KUKA KRL program: f1_Kuka_APT212T03S12.SRC

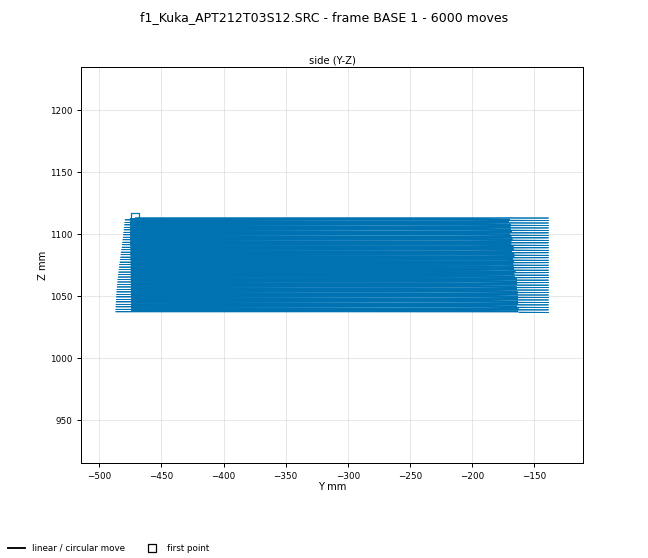
[picture p0: tool path of f1_Kuka_APT212T03S12.SRC in frame BASE 1, 6000 of 6001 moves have a stored position in this frame; points joined in program order, loops and branches not executed]
&ACCESS RVP
&REL 2
&PARAM TEMPLATE = C:\KRC\Roboter\Template\vorgabe
&PARAM EDITMASK = *
DEF f1_Kuka_APT212T03S12()


;FOLD INI;%{PE}%V3.2.0,%MKUKATPBASIS,%CINIT,%VCOMMON,%P
  ;FOLD BAS INI;%{E}%V3.2.0,%MKUKATPBASIS,%CINIT,%VINIT,%P
    GLOBAL INTERRUPT DECL 3 WHEN $STOPMESS==TRUE DO IR_STOPM ( )
    INTERRUPT ON 3
    BAS (#INITMOV,0 )
  ;ENDFOLD (BAS INI)
  ;FOLD USER INI;%{E}%V3.2.0,%MKUKATPUSER,%CINIT,%VINIT,%P
    ;Make your modifications here
  ;ENDFOLD (USER INI)
;ENDFOLD (INI)


;*** Make Null PTP Move
  PTP $pos_act

;*** Auto Load The Correct TOOL Data
  $tool=tool_data[3]

;*** Auto Load The Correct BASE Data
  $base=base_data[1]

  $ADVANCE = 5

;*** Restate Last Velocity
MMPM(30000.0)
SetRPM(6000)
LIN {X -0.139,Y -471.059,Z 1113.517,A 0.000,B 0.000,C 90.000,E1 273.151} C_DIS
LIN {X -0.055,Y -467.604,Z 1113.515,A 0.000,B 0.000,C 90.000,E1 272.636} C_DIS
LIN {X 0.015,Y -463.098,Z 1113.512,A 0.000,B 0.000,C 90.000,E1 272.121} C_DIS
LIN {X 0.076,Y -457.357,Z 1113.509,A 0.000,B 0.000,C 90.000,E1 271.604} C_DIS
LIN {X 0.094,Y -450.718,Z 1113.506,A 0.000,B 0.000,C 90.000,E1 271.146} C_DIS
LIN {X -0.014,Y -447.591,Z 1113.505,A 0.000,B 0.000,C 90.000,E1 270.974} C_DIS
LIN {X 0.034,Y -440.708,Z 1113.504,A 0.000,B 0.000,C 90.000,E1 270.630} C_DIS
LIN {X 0.083,Y -433.709,Z 1113.502,A 0.000,B 0.000,C 90.000,E1 270.344} C_DIS
LIN {X 0.062,Y -426.679,Z 1113.501,A 0.000,B 0.000,C 90.000,E1 270.115} C_DIS
LIN {X -0.084,Y -419.545,Z 1113.500,A 0.000,B 0.000,C 90.000,E1 269.943} C_DIS
LIN {X 0.009,Y -412.022,Z 1113.499,A 0.000,B 0.000,C 90.000,E1 269.771} C_DIS
LIN {X -0.097,Y -403.841,Z 1113.498,A 0.000,B 0.000,C 90.000,E1 269.656} C_DIS
LIN {X 0.016,Y -391.803,Z 1113.497,A 0.000,B 0.000,C 90.000,E1 269.542} C_DIS
LIN {X -0.051,Y -388.701,Z 1113.497,A 0.000,B 0.000,C 90.000,E1 269.542} C_DIS
LIN {X -0.056,Y -181.444,Z 1113.497,A 0.000,B 0.000,C 90.000,E1 269.542} C_DIS
LIN {X -0.018,Y -180.903,Z 1113.474,A 0.000,B 0.000,C 90.000,E1 265.298} C_DIS
LIN {X -0.068,Y -180.241,Z 1113.464,A 0.000,B 0.000,C 90.000,E1 263.628} C_DIS
LIN {X -0.049,Y -178.727,Z 1113.441,A 0.000,B 0.000,C 90.000,E1 259.398} C_DIS
LIN {X 0.018,Y -175.775,Z 1113.413,A 0.000,B 0.000,C 90.000,E1 254.283} C_DIS
LIN {X 0.006,Y -171.960,Z 1113.384,A 0.000,B 0.000,C 90.000,E1 249.156} C_DIS
LIN {X 0.044,Y -171.353,Z 1113.379,A 0.000,B 0.000,C 90.000,E1 248.284} C_DIS
LIN {X 0.021,Y -167.603,Z 1113.355,A 0.000,B 0.000,C 90.000,E1 243.973} C_DIS
LIN {X 0.034,Y -166.248,Z 1113.346,A 0.000,B 0.000,C 90.000,E1 242.231} C_DIS
LIN {X 0.021,Y -163.004,Z 1113.326,A 0.000,B 0.000,C 90.000,E1 238.742} C_DIS
LIN {X 0.068,Y -160.925,Z 1113.312,A 0.000,B 0.000,C 90.000,E1 236.087} C_DIS
LIN {X 0.045,Y -157.686,Z 1113.292,A 0.000,B 0.000,C 90.000,E1 232.557} C_DIS
LIN {X -0.016,Y -155.726,Z 1113.277,A 0.000,B 0.000,C 90.000,E1 229.908} C_DIS
LIN {X 0.037,Y -151.985,Z 1113.252,A 0.000,B 0.000,C 90.000,E1 225.405} C_DIS
LIN {X 0.053,Y -150.230,Z 1113.237,A 0.000,B 0.000,C 90.000,E1 222.690} C_DIS
LIN {X -0.024,Y -146.991,Z 1113.212,A 0.000,B 0.000,C 90.000,E1 218.177} C_DIS
LIN {X -0.033,Y -145.576,Z 1113.197,A 0.000,B 0.000,C 90.000,E1 215.438} C_DIS
LIN {X 0.083,Y -142.965,Z 1113.171,A 0.000,B 0.000,C 90.000,E1 210.797} C_DIS
LIN {X 0.013,Y -141.593,Z 1113.151,A 0.000,B 0.000,C 90.000,E1 207.129} C_DIS
LIN {X 0.061,Y -139.420,Z 1113.115,A 0.000,B 0.000,C 90.000,E1 200.610} C_DIS
LIN {X -0.019,Y -139.147,Z 1113.104,A 0.000,B 0.000,C 90.000,E1 198.779} C_DIS
LIN {X 0.003,Y -138.346,Z 1113.058,A 0.000,B 0.000,C 90.000,E1 190.366} C_DIS
LIN {X -0.011,Y -139.488,Z 1113.006,A 0.000,B 0.000,C 90.000,E1 181.031} C_DIS
LIN {X -0.071,Y -141.091,Z 1112.975,A 0.000,B 0.000,C 90.000,E1 175.469} C_DIS
LIN {X 0.023,Y -142.469,Z 1112.959,A 0.000,B 0.000,C 90.000,E1 172.648} C_DIS
LIN {X -0.029,Y -144.715,Z 1112.934,A 0.000,B 0.000,C 90.000,E1 168.049} C_DIS
LIN {X 0.064,Y -147.315,Z 1112.913,A 0.000,B 0.000,C 90.000,E1 164.338} C_DIS
LIN {X -0.063,Y -150.636,Z 1112.888,A 0.000,B 0.000,C 90.000,E1 159.826} C_DIS
LIN {X 0.012,Y -154.113,Z 1112.868,A 0.000,B 0.000,C 90.000,E1 156.177} C_DIS
LIN {X -0.064,Y -157.538,Z 1112.848,A 0.000,B 0.000,C 90.000,E1 152.615} C_DIS
LIN {X 0.101,Y -161.775,Z 1112.828,A 0.000,B 0.000,C 90.000,E1 148.997} C_DIS
LIN {X -0.014,Y -165.968,Z 1112.808,A 0.000,B 0.000,C 90.000,E1 145.515} C_DIS
LIN {X -0.019,Y -170.962,Z 1112.789,A 0.000,B 0.000,C 90.000,E1 142.029} C_DIS
LIN {X 0.033,Y -175.831,Z 1112.770,A 0.000,B 0.000,C 90.000,E1 138.566} C_DIS
LIN {X 0.028,Y -181.437,Z 1112.751,A 0.000,B 0.000,C 90.000,E1 135.162} C_DIS
LIN {X -0.098,Y -186.943,Z 1112.732,A 0.000,B 0.000,C 90.000,E1 131.838} C_DIS
LIN {X -0.100,Y -190.056,Z 1112.723,A 0.000,B 0.000,C 90.000,E1 130.172} C_DIS
LIN {X -0.085,Y -195.830,Z 1112.705,A 0.000,B 0.000,C 90.000,E1 126.870} C_DIS
LIN {X 0.022,Y -200.393,Z 1112.692,A 0.000,B 0.000,C 90.000,E1 124.532} C_DIS
LIN {X -0.001,Y -308.324,Z 1112.692,A 0.000,B 0.000,C 90.000,E1 124.532} C_DIS
LIN {X -0.072,Y -309.497,Z 1112.692,A 0.000,B 0.000,C 90.000,E1 124.532} C_DIS
LIN {X -0.028,Y -313.075,Z 1112.691,A 0.000,B 0.000,C 90.000,E1 124.405} C_DIS
LIN {X -0.040,Y -316.216,Z 1112.690,A 0.000,B 0.000,C 90.000,E1 124.199} C_DIS
LIN {X 0.038,Y -319.912,Z 1112.688,A 0.000,B 0.000,C 90.000,E1 123.785} C_DIS
LIN {X -0.021,Y -321.827,Z 1112.686,A 0.000,B 0.000,C 90.000,E1 123.499} C_DIS
LIN {X -0.081,Y -323.333,Z 1112.684,A 0.000,B 0.000,C 90.000,E1 123.214} C_DIS
LIN {X -0.084,Y -326.852,Z 1112.679,A 0.000,B 0.000,C 90.000,E1 122.260} C_DIS
LIN {X 0.052,Y -337.735,Z 1112.663,A 0.000,B 0.000,C 90.000,E1 119.411} C_DIS
LIN {X -0.122,Y -349.996,Z 1112.648,A 0.000,B 0.000,C 90.000,E1 116.668} C_DIS
LIN {X -0.116,Y -363.748,Z 1112.633,A 0.000,B 0.000,C 90.000,E1 113.951} C_DIS
LIN {X -0.114,Y -377.318,Z 1112.620,A 0.000,B 0.000,C 90.000,E1 111.589} C_DIS
LIN {X -0.044,Y -392.255,Z 1112.607,A 0.000,B 0.000,C 90.000,E1 109.268} C_DIS
LIN {X 0.158,Y -408.666,Z 1112.594,A 0.000,B 0.000,C 90.000,E1 106.985} C_DIS
LIN {X -0.146,Y -426.666,Z 1112.582,A 0.000,B 0.000,C 90.000,E1 104.828} C_DIS
LIN {X -0.136,Y -446.228,Z 1112.570,A 0.000,B 0.000,C 90.000,E1 102.703} C_DIS
LIN {X 0.014,Y -468.953,Z 1112.558,A 0.000,B 0.000,C 90.000,E1 100.489} C_DIS
LIN {X 0.041,Y -470.834,Z 1112.557,A 0.000,B 0.000,C 90.000,E1 100.254} C_DIS
LIN {X -0.107,Y -472.388,Z 1112.556,A 0.000,B 0.000,C 90.000,E1 100.018} C_DIS
LIN {X 0.211,Y -473.550,Z 1112.554,A 0.000,B 0.000,C 90.000,E1 99.726} C_DIS
LIN {X -0.147,Y -474.953,Z 1112.551,A 0.000,B 0.000,C 90.000,E1 99.265} C_DIS
LIN {X -0.026,Y -475.327,Z 1112.549,A 0.000,B 0.000,C 90.000,E1 98.746} C_DIS
LIN {X 0.173,Y -474.738,Z 1112.546,A 0.000,B 0.000,C 90.000,E1 98.219} C_DIS
LIN {X -0.166,Y -473.095,Z 1112.543,A 0.000,B 0.000,C 90.000,E1 97.757} C_DIS
LIN {X 0.102,Y -471.788,Z 1112.542,A 0.000,B 0.000,C 90.000,E1 97.473} C_DIS
LIN {X 0.009,Y -457.406,Z 1112.530,A 0.000,B 0.000,C 90.000,E1 95.454} C_DIS
LIN {X -0.050,Y -439.778,Z 1112.516,A 0.000,B 0.000,C 90.000,E1 92.865} C_DIS
LIN {X -0.072,Y -426.758,Z 1112.504,A 0.000,B 0.000,C 90.000,E1 90.745} C_DIS
LIN {X -0.028,Y -408.534,Z 1112.486,A 0.000,B 0.000,C 90.000,E1 87.478} C_DIS
LIN {X -0.013,Y -399.508,Z 1112.477,A 0.000,B 0.000,C 90.000,E1 85.812} C_DIS
LIN {X -0.106,Y -388.900,Z 1112.466,A 0.000,B 0.000,C 90.000,E1 83.856} C_DIS
LIN {X -0.001,Y -378.381,Z 1112.455,A 0.000,B 0.000,C 90.000,E1 81.837} C_DIS
LIN {X -0.006,Y -369.144,Z 1112.445,A 0.000,B 0.000,C 90.000,E1 80.095} C_DIS
LIN {X -0.108,Y -359.479,Z 1112.435,A 0.000,B 0.000,C 90.000,E1 78.342} C_DIS
LIN {X 0.042,Y -349.580,Z 1112.425,A 0.000,B 0.000,C 90.000,E1 76.520} C_DIS
LIN {X -0.003,Y -338.018,Z 1112.413,A 0.000,B 0.000,C 90.000,E1 74.393} C_DIS
LIN {X 0.018,Y -323.542,Z 1112.398,A 0.000,B 0.000,C 90.000,E1 71.583} C_DIS
LIN {X -0.047,Y -309.901,Z 1112.382,A 0.000,B 0.000,C 90.000,E1 68.720} C_DIS
LIN {X -0.139,Y -297.027,Z 1112.365,A 0.000,B 0.000,C 90.000,E1 65.793} C_DIS
LIN {X 0.053,Y -284.665,Z 1112.349,A 0.000,B 0.000,C 90.000,E1 62.743} C_DIS
LIN {X 0.089,Y -274.024,Z 1112.333,A 0.000,B 0.000,C 90.000,E1 59.999} C_DIS
LIN {X -0.096,Y -263.649,Z 1112.318,A 0.000,B 0.000,C 90.000,E1 57.248} C_DIS
LIN {X 0.013,Y -251.356,Z 1112.298,A 0.000,B 0.000,C 90.000,E1 53.657} C_DIS
LIN {X 0.084,Y -240.974,Z 1112.280,A 0.000,B 0.000,C 90.000,E1 50.356} C_DIS
LIN {X 0.013,Y -231.416,Z 1112.261,A 0.000,B 0.000,C 90.000,E1 47.025} C_DIS
LIN {X 0.072,Y -221.510,Z 1112.240,A 0.000,B 0.000,C 90.000,E1 43.218} C_DIS
LIN {X 0.029,Y -212.142,Z 1112.219,A 0.000,B 0.000,C 90.000,E1 39.358} C_DIS
LIN {X -0.011,Y -205.168,Z 1112.201,A 0.000,B 0.000,C 90.000,E1 36.217} C_DIS
LIN {X 0.026,Y -198.680,Z 1112.183,A 0.000,B 0.000,C 90.000,E1 33.007} C_DIS
LIN {X -0.084,Y -192.840,Z 1112.165,A 0.000,B 0.000,C 90.000,E1 29.795} C_DIS
LIN {X -0.018,Y -187.519,Z 1112.147,A 0.000,B 0.000,C 90.000,E1 26.488} C_DIS
LIN {X 0.012,Y -182.914,Z 1112.129,A 0.000,B 0.000,C 90.000,E1 23.153} C_DIS
LIN {X -0.046,Y -179.023,Z 1112.110,A 0.000,B 0.000,C 90.000,E1 19.812} C_DIS
LIN {X 0.012,Y -175.068,Z 1112.086,A 0.000,B 0.000,C 90.000,E1 15.552} C_DIS
LIN {X -0.065,Y -172.119,Z 1112.063,A 0.000,B 0.000,C 90.000,E1 11.299} C_DIS
LIN {X 0.069,Y -169.810,Z 1112.029,A 0.000,B 0.000,C 90.000,E1 5.220} C_DIS
LIN {X 0.050,Y -170.803,Z 1111.964,A 0.000,B 0.000,C 90.000,E1 353.457} C_DIS
LIN {X 0.054,Y -173.493,Z 1111.935,A 0.000,B 0.000,C 90.000,E1 348.285} C_DIS
LIN {X -0.029,Y -176.809,Z 1111.911,A 0.000,B 0.000,C 90.000,E1 344.031} C_DIS
LIN {X 0.071,Y -181.080,Z 1111.888,A 0.000,B 0.000,C 90.000,E1 339.752} C_DIS
LIN {X -0.005,Y -185.214,Z 1111.869,A 0.000,B 0.000,C 90.000,E1 336.410} C_DIS
LIN {X -0.007,Y -190.069,Z 1111.850,A 0.000,B 0.000,C 90.000,E1 333.076} C_DIS
LIN {X -0.055,Y -195.639,Z 1111.832,A 0.000,B 0.000,C 90.000,E1 329.793} C_DIS
LIN {X 0.072,Y -201.884,Z 1111.814,A 0.000,B 0.000,C 90.000,E1 326.501} C_DIS
LIN {X -0.094,Y -208.900,Z 1111.796,A 0.000,B 0.000,C 90.000,E1 323.336} C_DIS
LIN {X -0.005,Y -216.661,Z 1111.779,A 0.000,B 0.000,C 90.000,E1 320.150} C_DIS
LIN {X -0.078,Y -225.301,Z 1111.761,A 0.000,B 0.000,C 90.000,E1 317.067} C_DIS
LIN {X -0.102,Y -235.017,Z 1111.745,A 0.000,B 0.000,C 90.000,E1 314.028} C_DIS
LIN {X -0.003,Y -244.461,Z 1111.730,A 0.000,B 0.000,C 90.000,E1 311.391} C_DIS
LIN {X -0.029,Y -253.486,Z 1111.718,A 0.000,B 0.000,C 90.000,E1 309.197} C_DIS
LIN {X 0.046,Y -265.217,Z 1111.704,A 0.000,B 0.000,C 90.000,E1 306.664} C_DIS
LIN {X 0.120,Y -281.653,Z 1111.686,A 0.000,B 0.000,C 90.000,E1 303.499} C_DIS
LIN {X 0.046,Y -297.378,Z 1111.671,A 0.000,B 0.000,C 90.000,E1 300.797} C_DIS
LIN {X -0.029,Y -316.878,Z 1111.655,A 0.000,B 0.000,C 90.000,E1 297.847} C_DIS
LIN {X 0.057,Y -335.880,Z 1111.641,A 0.000,B 0.000,C 90.000,E1 295.283} C_DIS
LIN {X 0.015,Y -351.312,Z 1111.630,A 0.000,B 0.000,C 90.000,E1 293.462} C_DIS
LIN {X 0.107,Y -367.275,Z 1111.621,A 0.000,B 0.000,C 90.000,E1 291.770} C_DIS
LIN {X 0.039,Y -392.129,Z 1111.608,A 0.000,B 0.000,C 90.000,E1 289.504} C_DIS
LIN {X 0.001,Y -405.648,Z 1111.602,A 0.000,B 0.000,C 90.000,E1 288.308} C_DIS
LIN {X 0.092,Y -416.173,Z 1111.596,A 0.000,B 0.000,C 90.000,E1 287.330} C_DIS
LIN {X -0.150,Y -423.969,Z 1111.592,A 0.000,B 0.000,C 90.000,E1 286.622} C_DIS
LIN {X -0.028,Y -431.548,Z 1111.588,A 0.000,B 0.000,C 90.000,E1 285.843} C_DIS
LIN {X -0.081,Y -438.876,Z 1111.584,A 0.000,B 0.000,C 90.000,E1 285.064} C_DIS
LIN {X 0.109,Y -445.762,Z 1111.579,A 0.000,B 0.000,C 90.000,E1 284.245} C_DIS
LIN {X -0.063,Y -452.032,Z 1111.575,A 0.000,B 0.000,C 90.000,E1 283.480} C_DIS
LIN {X -0.088,Y -457.614,Z 1111.571,A 0.000,B 0.000,C 90.000,E1 282.703} C_DIS
LIN {X -0.261,Y -462.481,Z 1111.566,A 0.000,B 0.000,C 90.000,E1 281.951} C_DIS
LIN {X 0.159,Y -466.725,Z 1111.562,A 0.000,B 0.000,C 90.000,E1 281.130} C_DIS
LIN {X 0.163,Y -470.343,Z 1111.558,A 0.000,B 0.000,C 90.000,E1 280.366} C_DIS
LIN {X 0.109,Y -473.331,Z 1111.553,A 0.000,B 0.000,C 90.000,E1 279.613} C_DIS
LIN {X -0.253,Y -475.008,Z 1111.551,A 0.000,B 0.000,C 90.000,E1 279.151} C_DIS
LIN {X -0.062,Y -476.427,Z 1111.548,A 0.000,B 0.000,C 90.000,E1 278.624} C_DIS
LIN {X 0.068,Y -477.604,Z 1111.545,A 0.000,B 0.000,C 90.000,E1 278.106} C_DIS
LIN {X 0.208,Y -478.452,Z 1111.542,A 0.000,B 0.000,C 90.000,E1 277.587} C_DIS
LIN {X -0.118,Y -479.069,Z 1111.540,A 0.000,B 0.000,C 90.000,E1 277.125} C_DIS
LIN {X 0.037,Y -479.395,Z 1111.537,A 0.000,B 0.000,C 90.000,E1 276.606} C_DIS
LIN {X 0.195,Y -479.403,Z 1111.534,A 0.000,B 0.000,C 90.000,E1 276.087} C_DIS
LIN {X -0.122,Y -479.104,Z 1111.531,A 0.000,B 0.000,C 90.000,E1 275.625} C_DIS
LIN {X 0.037,Y -478.438,Z 1111.528,A 0.000,B 0.000,C 90.000,E1 275.106} C_DIS
LIN {X 0.191,Y -477.392,Z 1111.526,A 0.000,B 0.000,C 90.000,E1 274.588} C_DIS
LIN {X -0.170,Y -475.931,Z 1111.523,A 0.000,B 0.000,C 90.000,E1 274.131} C_DIS
LIN {X -0.027,Y -473.925,Z 1111.520,A 0.000,B 0.000,C 90.000,E1 273.612} C_DIS
LIN {X 0.103,Y -471.258,Z 1111.517,A 0.000,B 0.000,C 90.000,E1 273.094} C_DIS
LIN {X 0.187,Y -467.779,Z 1111.514,A 0.000,B 0.000,C 90.000,E1 272.579} C_DIS
LIN {X -0.011,Y -465.688,Z 1111.513,A 0.000,B 0.000,C 90.000,E1 272.350} C_DIS
LIN {X -0.207,Y -463.300,Z 1111.512,A 0.000,B 0.000,C 90.000,E1 272.121} C_DIS
LIN {X -0.142,Y -457.521,Z 1111.509,A 0.000,B 0.000,C 90.000,E1 271.604} C_DIS
LIN {X -0.080,Y -450.984,Z 1111.506,A 0.000,B 0.000,C 90.000,E1 271.146} C_DIS
LIN {X -0.200,Y -447.827,Z 1111.505,A 0.000,B 0.000,C 90.000,E1 270.974} C_DIS
LIN {X -0.172,Y -440.828,Z 1111.503,A 0.000,B 0.000,C 90.000,E1 270.630} C_DIS
LIN {X -0.140,Y -433.831,Z 1111.502,A 0.000,B 0.000,C 90.000,E1 270.344} C_DIS
LIN {X -0.148,Y -426.727,Z 1111.500,A 0.000,B 0.000,C 90.000,E1 270.115} C_DIS
LIN {X 0.155,Y -419.712,Z 1111.500,A 0.000,B 0.000,C 90.000,E1 269.885} C_DIS
LIN {X 0.185,Y -408.271,Z 1111.498,A 0.000,B 0.000,C 90.000,E1 269.656} C_DIS
LIN {X 0.035,Y -395.985,Z 1111.497,A 0.000,B 0.000,C 90.000,E1 269.542} C_DIS
LIN {X -0.169,Y -387.727,Z 1111.497,A 0.000,B 0.000,C 90.000,E1 269.542} C_DIS
LIN {X 0.071,Y -181.441,Z 1111.497,A 0.000,B 0.000,C 90.000,E1 269.484} C_DIS
LIN {X -0.073,Y -180.903,Z 1111.474,A 0.000,B 0.000,C 90.000,E1 265.298} C_DIS
LIN {X 0.057,Y -180.233,Z 1111.464,A 0.000,B 0.000,C 90.000,E1 263.571} C_DIS
LIN {X 0.072,Y -178.717,Z 1111.441,A 0.000,B 0.000,C 90.000,E1 259.342} C_DIS
LIN {X -0.035,Y -175.765,Z 1111.413,A 0.000,B 0.000,C 90.000,E1 254.283} C_DIS
LIN {X 0.014,Y -171.949,Z 1111.384,A 0.000,B 0.000,C 90.000,E1 249.135} C_DIS
LIN {X -0.009,Y -171.337,Z 1111.379,A 0.000,B 0.000,C 90.000,E1 248.284} C_DIS
LIN {X -0.031,Y -167.591,Z 1111.355,A 0.000,B 0.000,C 90.000,E1 243.973} C_DIS
LIN {X -0.018,Y -166.229,Z 1111.346,A 0.000,B 0.000,C 90.000,E1 242.231} C_DIS
LIN {X -0.030,Y -162.989,Z 1111.326,A 0.000,B 0.000,C 90.000,E1 238.742} C_DIS
LIN {X 0.017,Y -160.907,Z 1111.312,A 0.000,B 0.000,C 90.000,E1 236.087} C_DIS
LIN {X -0.005,Y -157.672,Z 1111.292,A 0.000,B 0.000,C 90.000,E1 232.557} C_DIS
LIN {X -0.067,Y -155.711,Z 1111.277,A 0.000,B 0.000,C 90.000,E1 229.908} C_DIS
LIN {X -0.013,Y -151.972,Z 1111.252,A 0.000,B 0.000,C 90.000,E1 225.405} C_DIS
LIN {X 0.005,Y -150.215,Z 1111.237,A 0.000,B 0.000,C 90.000,E1 222.690} C_DIS
LIN {X -0.072,Y -146.980,Z 1111.212,A 0.000,B 0.000,C 90.000,E1 218.177} C_DIS
LIN {X 0.037,Y -145.567,Z 1111.197,A 0.000,B 0.000,C 90.000,E1 215.391} C_DIS
LIN {X 0.037,Y -142.957,Z 1111.171,A 0.000,B 0.000,C 90.000,E1 210.797} C_DIS
LIN {X -0.033,Y -141.584,Z 1111.151,A 0.000,B 0.000,C 90.000,E1 207.129} C_DIS
LIN {X 0.014,Y -139.417,Z 1111.115,A 0.000,B 0.000,C 90.000,E1 200.610} C_DIS
LIN {X 0.067,Y -139.142,Z 1111.104,A 0.000,B 0.000,C 90.000,E1 198.725} C_DIS
LIN {X -0.043,Y -138.347,Z 1111.057,A 0.000,B 0.000,C 90.000,E1 190.366} C_DIS
LIN {X -0.058,Y -139.491,Z 1111.006,A 0.000,B 0.000,C 90.000,E1 181.031} C_DIS
LIN {X 0.023,Y -141.099,Z 1110.975,A 0.000,B 0.000,C 90.000,E1 175.412} C_DIS
LIN {X -0.024,Y -142.479,Z 1110.959,A 0.000,B 0.000,C 90.000,E1 172.648} C_DIS
LIN {X 0.065,Y -144.727,Z 1110.933,A 0.000,B 0.000,C 90.000,E1 167.993} C_DIS
LIN {X 0.016,Y -147.330,Z 1110.913,A 0.000,B 0.000,C 90.000,E1 164.338} C_DIS
LIN {X 0.081,Y -150.652,Z 1110.888,A 0.000,B 0.000,C 90.000,E1 159.752} C_DIS
LIN {X -0.037,Y -154.130,Z 1110.868,A 0.000,B 0.000,C 90.000,E1 156.177} C_DIS
LIN {X 0.025,Y -157.557,Z 1110.848,A 0.000,B 0.000,C 90.000,E1 152.564} C_DIS
LIN {X 0.050,Y -161.799,Z 1110.828,A 0.000,B 0.000,C 90.000,E1 148.997} C_DIS
LIN {X 0.070,Y -165.990,Z 1110.808,A 0.000,B 0.000,C 90.000,E1 145.468} C_DIS
LIN {X 0.063,Y -170.989,Z 1110.789,A 0.000,B 0.000,C 90.000,E1 141.984} C_DIS
LIN {X -0.021,Y -175.857,Z 1110.770,A 0.000,B 0.000,C 90.000,E1 138.566} C_DIS
LIN {X -0.027,Y -181.463,Z 1110.751,A 0.000,B 0.000,C 90.000,E1 135.162} C_DIS
LIN {X 0.110,Y -186.974,Z 1110.732,A 0.000,B 0.000,C 90.000,E1 131.757} C_DIS
LIN {X 0.112,Y -190.088,Z 1110.723,A 0.000,B 0.000,C 90.000,E1 130.092} C_DIS
LIN {X 0.015,Y -195.861,Z 1110.705,A 0.000,B 0.000,C 90.000,E1 126.824} C_DIS
LIN {X 0.017,Y -200.329,Z 1110.692,A 0.000,B 0.000,C 90.000,E1 124.565} C_DIS
LIN {X 0.166,Y -307.637,Z 1110.692,A 0.000,B 0.000,C 90.000,E1 124.532} C_DIS
LIN {X 0.131,Y -308.781,Z 1110.692,A 0.000,B 0.000,C 90.000,E1 124.532} C_DIS
LIN {X -0.118,Y -313.804,Z 1110.691,A 0.000,B 0.000,C 90.000,E1 124.405} C_DIS
LIN {X -0.174,Y -316.709,Z 1110.690,A 0.000,B 0.000,C 90.000,E1 124.199} C_DIS
LIN {X 0.113,Y -320.458,Z 1110.687,A 0.000,B 0.000,C 90.000,E1 123.706} C_DIS
LIN {X -0.049,Y -322.322,Z 1110.686,A 0.000,B 0.000,C 90.000,E1 123.420} C_DIS
LIN {X 0.056,Y -323.778,Z 1110.684,A 0.000,B 0.000,C 90.000,E1 123.086} C_DIS
LIN {X 0.082,Y -336.846,Z 1110.665,A 0.000,B 0.000,C 90.000,E1 119.617} C_DIS
LIN {X -0.115,Y -349.001,Z 1110.649,A 0.000,B 0.000,C 90.000,E1 116.873} C_DIS
LIN {X 0.024,Y -362.634,Z 1110.634,A 0.000,B 0.000,C 90.000,E1 114.131} C_DIS
LIN {X 0.000,Y -376.093,Z 1110.621,A 0.000,B 0.000,C 90.000,E1 111.770} C_DIS
LIN {X 0.040,Y -390.910,Z 1110.608,A 0.000,B 0.000,C 90.000,E1 109.450} C_DIS
LIN {X -0.178,Y -407.190,Z 1110.596,A 0.000,B 0.000,C 90.000,E1 107.221} C_DIS
LIN {X -0.123,Y -425.050,Z 1110.583,A 0.000,B 0.000,C 90.000,E1 105.009} C_DIS
LIN {X -0.179,Y -444.502,Z 1110.571,A 0.000,B 0.000,C 90.000,E1 102.883} C_DIS
LIN {X -0.085,Y -464.739,Z 1110.560,A 0.000,B 0.000,C 90.000,E1 100.894} C_DIS
LIN {X -0.060,Y -469.593,Z 1110.558,A 0.000,B 0.000,C 90.000,E1 100.423} C_DIS
LIN {X -0.111,Y -471.308,Z 1110.557,A 0.000,B 0.000,C 90.000,E1 100.197} C_DIS
LIN {X 0.209,Y -472.734,Z 1110.555,A 0.000,B 0.000,C 90.000,E1 99.905} C_DIS
LIN {X 0.063,Y -473.796,Z 1110.554,A 0.000,B 0.000,C 90.000,E1 99.670} C_DIS
LIN {X 0.176,Y -475.035,Z 1110.551,A 0.000,B 0.000,C 90.000,E1 99.151} C_DIS
LIN {X -0.098,Y -475.268,Z 1110.548,A 0.000,B 0.000,C 90.000,E1 98.681} C_DIS
LIN {X 0.029,Y -474.534,Z 1110.545,A 0.000,B 0.000,C 90.000,E1 98.163} C_DIS
LIN {X 0.161,Y -472.714,Z 1110.543,A 0.000,B 0.000,C 90.000,E1 97.644} C_DIS
LIN {X 0.022,Y -471.293,Z 1110.541,A 0.000,B 0.000,C 90.000,E1 97.409} C_DIS
LIN {X -0.094,Y -456.843,Z 1110.530,A 0.000,B 0.000,C 90.000,E1 95.391} C_DIS
LIN {X 0.057,Y -440.932,Z 1110.517,A 0.000,B 0.000,C 90.000,E1 93.037} C_DIS
LIN {X 0.056,Y -427.874,Z 1110.505,A 0.000,B 0.000,C 90.000,E1 90.917} C_DIS
LIN {X -0.147,Y -413.962,Z 1110.492,A 0.000,B 0.000,C 90.000,E1 88.511} C_DIS
LIN {X -0.039,Y -405.097,Z 1110.482,A 0.000,B 0.000,C 90.000,E1 86.846} C_DIS
LIN {X -0.047,Y -394.489,Z 1110.472,A 0.000,B 0.000,C 90.000,E1 84.894} C_DIS
LIN {X 0.162,Y -382.415,Z 1110.459,A 0.000,B 0.000,C 90.000,E1 82.591} C_DIS
LIN {X -0.146,Y -373.276,Z 1110.449,A 0.000,B 0.000,C 90.000,E1 80.905} C_DIS
LIN {X 0.138,Y -365.409,Z 1110.441,A 0.000,B 0.000,C 90.000,E1 79.398} C_DIS
LIN {X 0.007,Y -357.267,Z 1110.433,A 0.000,B 0.000,C 90.000,E1 77.937} C_DIS
LIN {X 0.032,Y -345.686,Z 1110.421,A 0.000,B 0.000,C 90.000,E1 75.825} C_DIS
LIN {X -0.016,Y -334.165,Z 1110.409,A 0.000,B 0.000,C 90.000,E1 73.685} C_DIS
LIN {X -0.059,Y -318.384,Z 1110.392,A 0.000,B 0.000,C 90.000,E1 70.550} C_DIS
LIN {X 0.050,Y -302.190,Z 1110.372,A 0.000,B 0.000,C 90.000,E1 66.975} C_DIS
LIN {X -0.127,Y -289.617,Z 1110.356,A 0.000,B 0.000,C 90.000,E1 64.024} C_DIS
LIN {X 0.106,Y -277.484,Z 1110.339,A 0.000,B 0.000,C 90.000,E1 60.923} C_DIS
LIN {X -0.135,Y -266.989,Z 1110.323,A 0.000,B 0.000,C 90.000,E1 58.201} C_DIS
LIN {X 0.084,Y -254.446,Z 1110.303,A 0.000,B 0.000,C 90.000,E1 54.609} C_DIS
LIN {X -0.049,Y -243.833,Z 1110.285,A 0.000,B 0.000,C 90.000,E1 51.376} C_DIS
LIN {X 0.011,Y -235.060,Z 1110.269,A 0.000,B 0.000,C 90.000,E1 48.405} C_DIS
LIN {X -0.128,Y -224.893,Z 1110.248,A 0.000,B 0.000,C 90.000,E1 44.676} C_DIS
LIN {X -0.079,Y -217.174,Z 1110.231,A 0.000,B 0.000,C 90.000,E1 41.595} C_DIS
LIN {X -0.024,Y -209.844,Z 1110.214,A 0.000,B 0.000,C 90.000,E1 38.463} C_DIS
LIN {X -0.079,Y -202.993,Z 1110.196,A 0.000,B 0.000,C 90.000,E1 35.311} C_DIS
LIN {X -0.035,Y -196.666,Z 1110.178,A 0.000,B 0.000,C 90.000,E1 32.084} C_DIS
LIN {X -0.019,Y -190.939,Z 1110.160,A 0.000,B 0.000,C 90.000,E1 28.821} C_DIS
LIN {X -0.081,Y -185.840,Z 1110.142,A 0.000,B 0.000,C 90.000,E1 25.540} C_DIS
LIN {X 0.076,Y -181.426,Z 1110.123,A 0.000,B 0.000,C 90.000,E1 22.153} C_DIS
LIN {X 0.036,Y -176.914,Z 1110.100,A 0.000,B 0.000,C 90.000,E1 17.946} C_DIS
LIN {X -0.020,Y -173.388,Z 1110.076,A 0.000,B 0.000,C 90.000,E1 13.703} C_DIS
LIN {X 0.087,Y -170.557,Z 1110.047,A 0.000,B 0.000,C 90.000,E1 8.511} C_DIS
LIN {X 0.055,Y -171.265,Z 1109.954,A 0.000,B 0.000,C 90.000,E1 351.724} C_DIS
LIN {X -0.032,Y -174.411,Z 1109.925,A 0.000,B 0.000,C 90.000,E1 346.589} C_DIS
LIN {X -0.003,Y -178.106,Z 1109.902,A 0.000,B 0.000,C 90.000,E1 342.308} C_DIS
LIN {X -0.093,Y -182.777,Z 1109.878,A 0.000,B 0.000,C 90.000,E1 338.103} C_DIS
LIN {X 0.012,Y -187.295,Z 1109.859,A 0.000,B 0.000,C 90.000,E1 334.717} C_DIS
LIN {X 0.057,Y -192.501,Z 1109.841,A 0.000,B 0.000,C 90.000,E1 331.385} C_DIS
LIN {X 0.003,Y -198.430,Z 1109.823,A 0.000,B 0.000,C 90.000,E1 328.122} C_DIS
LIN {X -0.027,Y -205.094,Z 1109.805,A 0.000,B 0.000,C 90.000,E1 324.895} C_DIS
LIN {X 0.007,Y -212.486,Z 1109.787,A 0.000,B 0.000,C 90.000,E1 321.698} C_DIS
LIN {X 0.001,Y -220.669,Z 1109.770,A 0.000,B 0.000,C 90.000,E1 318.566} C_DIS
LIN {X 0.021,Y -229.863,Z 1109.753,A 0.000,B 0.000,C 90.000,E1 315.486} C_DIS
LIN {X 0.124,Y -240.139,Z 1109.736,A 0.000,B 0.000,C 90.000,E1 312.447} C_DIS
LIN {X 0.023,Y -250.245,Z 1109.722,A 0.000,B 0.000,C 90.000,E1 309.886} C_DIS
LIN {X -0.019,Y -261.690,Z 1109.708,A 0.000,B 0.000,C 90.000,E1 307.363} C_DIS
LIN {X 0.008,Y -275.993,Z 1109.692,A 0.000,B 0.000,C 90.000,E1 304.532} C_DIS
LIN {X -0.081,Y -293.364,Z 1109.675,A 0.000,B 0.000,C 90.000,E1 301.465} C_DIS
LIN {X -0.166,Y -310.239,Z 1109.660,A 0.000,B 0.000,C 90.000,E1 298.821} C_DIS
LIN {X -0.116,Y -328.605,Z 1109.646,A 0.000,B 0.000,C 90.000,E1 296.232} C_DIS
LIN {X 0.039,Y -343.557,Z 1109.635,A 0.000,B 0.000,C 90.000,E1 294.335} C_DIS
LIN {X -0.035,Y -359.326,Z 1109.625,A 0.000,B 0.000,C 90.000,E1 292.589} C_DIS
LIN {X 0.034,Y -372.860,Z 1109.618,A 0.000,B 0.000,C 90.000,E1 291.227} C_DIS
LIN {X 0.077,Y -391.938,Z 1109.608,A 0.000,B 0.000,C 90.000,E1 289.504} C_DIS
LIN {X 0.024,Y -405.532,Z 1109.602,A 0.000,B 0.000,C 90.000,E1 288.308} C_DIS
LIN {X 0.038,Y -416.005,Z 1109.596,A 0.000,B 0.000,C 90.000,E1 287.347} C_DIS
LIN {X -0.023,Y -423.765,Z 1109.592,A 0.000,B 0.000,C 90.000,E1 286.622} C_DIS
LIN {X -0.027,Y -433.789,Z 1109.587,A 0.000,B 0.000,C 90.000,E1 285.607} C_DIS
LIN {X -0.067,Y -440.969,Z 1109.582,A 0.000,B 0.000,C 90.000,E1 284.828} C_DIS
LIN {X 0.146,Y -447.690,Z 1109.578,A 0.000,B 0.000,C 90.000,E1 284.008} C_DIS
LIN {X -0.016,Y -453.840,Z 1109.574,A 0.000,B 0.000,C 90.000,E1 283.244} C_DIS
LIN {X -0.119,Y -459.210,Z 1109.569,A 0.000,B 0.000,C 90.000,E1 282.479} C_DIS
LIN {X -0.183,Y -463.924,Z 1109.565,A 0.000,B 0.000,C 90.000,E1 281.715} C_DIS
LIN {X -0.205,Y -468.000,Z 1109.561,A 0.000,B 0.000,C 90.000,E1 280.950} C_DIS
LIN {X 0.181,Y -471.437,Z 1109.557,A 0.000,B 0.000,C 90.000,E1 280.141} C_DIS
LIN {X -0.105,Y -473.383,Z 1109.554,A 0.000,B 0.000,C 90.000,E1 279.670} C_DIS
LIN {X 0.000,Y -475.083,Z 1109.551,A 0.000,B 0.000,C 90.000,E1 279.151} C_DIS
LIN {X 0.193,Y -476.504,Z 1109.548,A 0.000,B 0.000,C 90.000,E1 278.624} C_DIS
LIN {X -0.150,Y -477.683,Z 1109.545,A 0.000,B 0.000,C 90.000,E1 278.163} C_DIS
LIN {X -0.010,Y -478.581,Z 1109.542,A 0.000,B 0.000,C 90.000,E1 277.644} C_DIS
LIN {X 0.139,Y -479.234,Z 1109.540,A 0.000,B 0.000,C 90.000,E1 277.125} C_DIS
LIN {X -0.181,Y -479.586,Z 1109.537,A 0.000,B 0.000,C 90.000,E1 276.663} C_DIS
LIN {X -0.023,Y -479.630,Z 1109.534,A 0.000,B 0.000,C 90.000,E1 276.144} C_DIS
LIN {X 0.138,Y -479.374,Z 1109.531,A 0.000,B 0.000,C 90.000,E1 275.625} C_DIS
LIN {X -0.179,Y -478.763,Z 1109.529,A 0.000,B 0.000,C 90.000,E1 275.163} C_DIS
LIN {X -0.023,Y -477.810,Z 1109.526,A 0.000,B 0.000,C 90.000,E1 274.645} C_DIS
LIN {X 0.093,Y -476.351,Z 1109.523,A 0.000,B 0.000,C 90.000,E1 274.131} C_DIS
LIN {X -0.236,Y -474.412,Z 1109.520,A 0.000,B 0.000,C 90.000,E1 273.669} C_DIS
LIN {X -0.128,Y -471.831,Z 1109.517,A 0.000,B 0.000,C 90.000,E1 273.154} C_DIS
LIN {X 0.176,Y -470.299,Z 1109.516,A 0.000,B 0.000,C 90.000,E1 272.865} C_DIS
LIN {X -0.209,Y -466.403,Z 1109.513,A 0.000,B 0.000,C 90.000,E1 272.407} C_DIS
LIN {X 0.060,Y -464.086,Z 1109.512,A 0.000,B 0.000,C 90.000,E1 272.121} C_DIS
LIN {X -0.143,Y -461.462,Z 1109.510,A 0.000,B 0.000,C 90.000,E1 271.892} C_DIS
LIN {X 0.185,Y -455.473,Z 1109.508,A 0.000,B 0.000,C 90.000,E1 271.375} C_DIS
LIN {X 0.084,Y -449.127,Z 1109.505,A 0.000,B 0.000,C 90.000,E1 270.974} C_DIS
LIN {X 0.048,Y -442.260,Z 1109.504,A 0.000,B 0.000,C 90.000,E1 270.630} C_DIS
LIN {X 0.014,Y -435.268,Z 1109.502,A 0.000,B 0.000,C 90.000,E1 270.344} C_DIS
LIN {X -0.098,Y -427.919,Z 1109.501,A 0.000,B 0.000,C 90.000,E1 270.115} C_DIS
LIN {X 0.130,Y -420.709,Z 1109.500,A 0.000,B 0.000,C 90.000,E1 269.885} C_DIS
LIN {X -0.187,Y -413.154,Z 1109.499,A 0.000,B 0.000,C 90.000,E1 269.771} C_DIS
LIN {X 0.137,Y -405.236,Z 1109.498,A 0.000,B 0.000,C 90.000,E1 269.599} C_DIS
LIN {X -0.144,Y -394.039,Z 1109.497,A 0.000,B 0.000,C 90.000,E1 269.542} C_DIS
LIN {X 0.108,Y -387.694,Z 1109.497,A 0.000,B 0.000,C 90.000,E1 269.484} C_DIS
LIN {X 0.019,Y -181.436,Z 1109.497,A 0.000,B 0.000,C 90.000,E1 269.484} C_DIS
LIN {X -0.041,Y -180.846,Z 1109.472,A 0.000,B 0.000,C 90.000,E1 264.951} C_DIS
LIN {X 0.042,Y -178.956,Z 1109.444,A 0.000,B 0.000,C 90.000,E1 259.859} C_DIS
LIN {X -0.066,Y -177.358,Z 1109.430,A 0.000,B 0.000,C 90.000,E1 257.353} C_DIS
LIN {X 0.030,Y -175.529,Z 1109.411,A 0.000,B 0.000,C 90.000,E1 253.921} C_DIS
LIN {X 0.032,Y -172.265,Z 1109.387,A 0.000,B 0.000,C 90.000,E1 249.645} C_DIS
LIN {X 0.070,Y -171.744,Z 1109.382,A 0.000,B 0.000,C 90.000,E1 248.773} C_DIS
LIN {X -0.072,Y -167.341,Z 1109.353,A 0.000,B 0.000,C 90.000,E1 243.640} C_DIS
LIN {X 0.010,Y -166.727,Z 1109.349,A 0.000,B 0.000,C 90.000,E1 242.743} C_DIS
LIN {X -0.077,Y -162.707,Z 1109.324,A 0.000,B 0.000,C 90.000,E1 238.408} C_DIS
LIN {X -0.016,Y -161.398,Z 1109.315,A 0.000,B 0.000,C 90.000,E1 236.628} C_DIS
LIN {X 0.026,Y -157.391,Z 1109.290,A 0.000,B 0.000,C 90.000,E1 232.190} C_DIS
LIN {X -0.040,Y -155.388,Z 1109.275,A 0.000,B 0.000,C 90.000,E1 229.542} C_DIS
LIN {X 0.000,Y -151.722,Z 1109.250,A 0.000,B 0.000,C 90.000,E1 225.040} C_DIS
LIN {X 0.016,Y -149.916,Z 1109.235,A 0.000,B 0.000,C 90.000,E1 222.324} C_DIS
LIN {X -0.066,Y -146.771,Z 1109.210,A 0.000,B 0.000,C 90.000,E1 217.810} C_DIS
LIN {X 0.037,Y -145.340,Z 1109.195,A 0.000,B 0.000,C 90.000,E1 215.025} C_DIS
LIN {X -0.048,Y -142.418,Z 1109.164,A 0.000,B 0.000,C 90.000,E1 209.539} C_DIS
LIN {X 0.002,Y -141.403,Z 1109.149,A 0.000,B 0.000,C 90.000,E1 206.744} C_DIS
LIN {X -0.010,Y -139.356,Z 1109.112,A 0.000,B 0.000,C 90.000,E1 200.248} C_DIS
LIN {X -0.023,Y -138.797,Z 1109.097,A 0.000,B 0.000,C 90.000,E1 197.457} C_DIS
LIN {X 0.032,Y -138.347,Z 1109.055,A 0.000,B 0.000,C 90.000,E1 189.962} C_DIS
LIN {X 0.050,Y -139.373,Z 1109.009,A 0.000,B 0.000,C 90.000,E1 181.547} C_DIS
LIN {X -0.037,Y -141.262,Z 1108.973,A 0.000,B 0.000,C 90.000,E1 175.065} C_DIS
LIN {X 0.063,Y -142.629,Z 1108.957,A 0.000,B 0.000,C 90.000,E1 172.243} C_DIS
LIN {X 0.014,Y -144.954,Z 1108.931,A 0.000,B 0.000,C 90.000,E1 167.645} C_DIS
LIN {X 0.006,Y -147.582,Z 1108.911,A 0.000,B 0.000,C 90.000,E1 163.976} C_DIS
LIN {X 0.035,Y -150.195,Z 1108.891,A 0.000,B 0.000,C 90.000,E1 160.315} C_DIS
LIN {X -0.037,Y -153.577,Z 1108.871,A 0.000,B 0.000,C 90.000,E1 156.719} C_DIS
LIN {X -0.047,Y -156.993,Z 1108.851,A 0.000,B 0.000,C 90.000,E1 153.127} C_DIS
LIN {X 0.026,Y -161.108,Z 1108.831,A 0.000,B 0.000,C 90.000,E1 149.537} C_DIS
LIN {X -0.030,Y -163.211,Z 1108.821,A 0.000,B 0.000,C 90.000,E1 147.788} C_DIS
LIN {X -0.025,Y -167.639,Z 1108.802,A 0.000,B 0.000,C 90.000,E1 144.276} C_DIS
LIN {X -0.010,Y -171.464,Z 1108.787,A 0.000,B 0.000,C 90.000,E1 141.662} C_DIS
LIN {X -0.079,Y -176.391,Z 1108.768,A 0.000,B 0.000,C 90.000,E1 138.243} C_DIS
LIN {X 0.042,Y -180.684,Z 1108.754,A 0.000,B 0.000,C 90.000,E1 135.648} C_DIS
LIN {X 0.024,Y -186.086,Z 1108.735,A 0.000,B 0.000,C 90.000,E1 132.285} C_DIS
LIN {X -0.039,Y -190.723,Z 1108.721,A 0.000,B 0.000,C 90.000,E1 129.806} C_DIS
LIN {X -0.007,Y -196.477,Z 1108.703,A 0.000,B 0.000,C 90.000,E1 126.503} C_DIS
LIN {X -0.086,Y -200.293,Z 1108.692,A 0.000,B 0.000,C 90.000,E1 124.612} C_DIS
LIN {X -0.180,Y -308.479,Z 1108.692,A 0.000,B 0.000,C 90.000,E1 124.612} C_DIS
LIN {X 0.108,Y -310.100,Z 1108.692,A 0.000,B 0.000,C 90.000,E1 124.532} C_DIS
LIN {X -0.109,Y -315.207,Z 1108.691,A 0.000,B 0.000,C 90.000,E1 124.326} C_DIS
LIN {X -0.066,Y -317.925,Z 1108.689,A 0.000,B 0.000,C 90.000,E1 124.072} C_DIS
LIN {X -0.211,Y -321.649,Z 1108.686,A 0.000,B 0.000,C 90.000,E1 123.579} C_DIS
LIN {X 0.041,Y -323.250,Z 1108.685,A 0.000,B 0.000,C 90.000,E1 123.214} C_DIS
LIN {X -0.112,Y -330.216,Z 1108.674,A 0.000,B 0.000,C 90.000,E1 121.337} C_DIS
LIN {X 0.127,Y -341.537,Z 1108.658,A 0.000,B 0.000,C 90.000,E1 118.487} C_DIS
LIN {X -0.103,Y -354.271,Z 1108.643,A 0.000,B 0.000,C 90.000,E1 115.771} C_DIS
LIN {X -0.123,Y -368.535,Z 1108.628,A 0.000,B 0.000,C 90.000,E1 113.078} C_DIS
LIN {X -0.139,Y -382.594,Z 1108.615,A 0.000,B 0.000,C 90.000,E1 110.737} C_DIS
LIN {X 0.067,Y -398.060,Z 1108.602,A 0.000,B 0.000,C 90.000,E1 108.417} C_DIS
LIN {X -0.097,Y -415.040,Z 1108.590,A 0.000,B 0.000,C 90.000,E1 106.205} C_DIS
LIN {X 0.048,Y -433.655,Z 1108.578,A 0.000,B 0.000,C 90.000,E1 104.008} C_DIS
LIN {X -0.059,Y -453.575,Z 1108.566,A 0.000,B 0.000,C 90.000,E1 101.951} C_DIS
LIN {X 0.104,Y -468.790,Z 1108.558,A 0.000,B 0.000,C 90.000,E1 100.489} C_DIS
LIN {X 0.075,Y -470.744,Z 1108.557,A 0.000,B 0.000,C 90.000,E1 100.254} C_DIS
LIN {X 0.044,Y -472.230,Z 1108.556,A 0.000,B 0.000,C 90.000,E1 100.018} C_DIS
LIN {X -0.180,Y -473.414,Z 1108.554,A 0.000,B 0.000,C 90.000,E1 99.792} C_DIS
LIN {X 0.145,Y -474.277,Z 1108.553,A 0.000,B 0.000,C 90.000,E1 99.500} C_DIS
LIN {X -0.130,Y -475.186,Z 1108.550,A 0.000,B 0.000,C 90.000,E1 99.029} C_DIS
LIN {X -0.007,Y -475.115,Z 1108.547,A 0.000,B 0.000,C 90.000,E1 98.511} C_DIS
LIN {X 0.125,Y -474.060,Z 1108.544,A 0.000,B 0.000,C 90.000,E1 97.992} C_DIS
LIN {X -0.012,Y -473.117,Z 1108.543,A 0.000,B 0.000,C 90.000,E1 97.757} C_DIS
LIN {X -0.211,Y -471.839,Z 1108.542,A 0.000,B 0.000,C 90.000,E1 97.530} C_DIS
LIN {X 0.223,Y -466.415,Z 1108.537,A 0.000,B 0.000,C 90.000,E1 96.720} C_DIS
LIN {X 0.197,Y -453.842,Z 1108.528,A 0.000,B 0.000,C 90.000,E1 94.935} C_DIS
LIN {X 0.096,Y -439.840,Z 1108.516,A 0.000,B 0.000,C 90.000,E1 92.865} C_DIS
LIN {X 0.070,Y -426.818,Z 1108.504,A 0.000,B 0.000,C 90.000,E1 90.745} C_DIS
LIN {X 0.028,Y -410.068,Z 1108.488,A 0.000,B 0.000,C 90.000,E1 87.764} C_DIS
LIN {X 0.044,Y -401.083,Z 1108.478,A 0.000,B 0.000,C 90.000,E1 86.102} C_DIS
LIN {X -0.025,Y -390.442,Z 1108.467,A 0.000,B 0.000,C 90.000,E1 84.147} C_DIS
LIN {X 0.105,Y -379.916,Z 1108.456,A 0.000,B 0.000,C 90.000,E1 82.129} C_DIS
LIN {X 0.121,Y -370.667,Z 1108.447,A 0.000,B 0.000,C 90.000,E1 80.387} C_DIS
LIN {X 0.069,Y -362.686,Z 1108.439,A 0.000,B 0.000,C 90.000,E1 78.926} C_DIS
LIN {X -0.148,Y -352.821,Z 1108.429,A 0.000,B 0.000,C 90.000,E1 77.173} C_DIS
LIN {X -0.126,Y -341.225,Z 1108.417,A 0.000,B 0.000,C 90.000,E1 75.046} C_DIS
LIN {X 0.025,Y -328.213,Z 1108.403,A 0.000,B 0.000,C 90.000,E1 72.543} C_DIS
LIN {X -0.017,Y -314.308,Z 1108.387,A 0.000,B 0.000,C 90.000,E1 69.699} C_DIS
LIN {X 0.063,Y -299.815,Z 1108.369,A 0.000,B 0.000,C 90.000,E1 66.433} C_DIS
LIN {X -0.070,Y -287.283,Z 1108.353,A 0.000,B 0.000,C 90.000,E1 63.461} C_DIS
LIN {X 0.031,Y -276.533,Z 1108.337,A 0.000,B 0.000,C 90.000,E1 60.717} C_DIS
LIN {X 0.077,Y -267.349,Z 1108.324,A 0.000,B 0.000,C 90.000,E1 58.280} C_DIS
LIN {X -0.063,Y -254.743,Z 1108.304,A 0.000,B 0.000,C 90.000,E1 54.769} C_DIS
LIN {X -0.001,Y -244.072,Z 1108.286,A 0.000,B 0.000,C 90.000,E1 51.492} C_DIS
LIN {X 0.006,Y -234.198,Z 1108.268,A 0.000,B 0.000,C 90.000,E1 48.162} C_DIS
LIN {X -0.035,Y -226.037,Z 1108.251,A 0.000,B 0.000,C 90.000,E1 45.162} C_DIS
LIN {X 0.043,Y -218.223,Z 1108.234,A 0.000,B 0.000,C 90.000,E1 42.081} C_DIS
LIN {X -0.038,Y -210.812,Z 1108.217,A 0.000,B 0.000,C 90.000,E1 38.991} C_DIS
LIN {X 0.055,Y -203.853,Z 1108.199,A 0.000,B 0.000,C 90.000,E1 35.804} C_DIS
LIN {X -0.048,Y -197.409,Z 1108.181,A 0.000,B 0.000,C 90.000,E1 32.625} C_DIS
LIN {X 0.082,Y -191.575,Z 1108.163,A 0.000,B 0.000,C 90.000,E1 29.333} C_DIS
LIN {X 0.028,Y -186.352,Z 1108.145,A 0.000,B 0.000,C 90.000,E1 26.052} C_DIS
LIN {X 0.032,Y -181.843,Z 1108.126,A 0.000,B 0.000,C 90.000,E1 22.717} C_DIS
LIN {X 0.053,Y -178.027,Z 1108.108,A 0.000,B 0.000,C 90.000,E1 19.341} C_DIS
LIN {X -0.081,Y -174.175,Z 1108.084,A 0.000,B 0.000,C 90.000,E1 15.134} C_DIS
LIN {X -0.005,Y -170.946,Z 1108.055,A 0.000,B 0.000,C 90.000,E1 9.962} C_DIS
LIN {X 0.001,Y -168.831,Z 1108.012,A 0.000,B 0.000,C 90.000,E1 2.178} C_DIS
LIN {X 0.027,Y -170.256,Z 1107.964,A 0.000,B 0.000,C 90.000,E1 353.457} C_DIS
LIN {X 0.011,Y -172.909,Z 1107.935,A 0.000,B 0.000,C 90.000,E1 348.285} C_DIS
LIN {X 0.079,Y -176.190,Z 1107.911,A 0.000,B 0.000,C 90.000,E1 343.976} C_DIS
LIN {X -0.011,Y -180.487,Z 1107.887,A 0.000,B 0.000,C 90.000,E1 339.752} C_DIS
LIN {X 0.065,Y -184.653,Z 1107.869,A 0.000,B 0.000,C 90.000,E1 336.357} C_DIS
LIN {X -0.037,Y -189.523,Z 1107.850,A 0.000,B 0.000,C 90.000,E1 333.050} C_DIS
LIN {X -0.019,Y -195.137,Z 1107.832,A 0.000,B 0.000,C 90.000,E1 329.744} C_DIS
LIN {X -0.077,Y -201.457,Z 1107.814,A 0.000,B 0.000,C 90.000,E1 326.501} C_DIS
LIN {X 0.032,Y -208.472,Z 1107.796,A 0.000,B 0.000,C 90.000,E1 323.256} C_DIS
LIN {X -0.042,Y -216.303,Z 1107.778,A 0.000,B 0.000,C 90.000,E1 320.114} C_DIS
LIN {X 0.041,Y -224.957,Z 1107.761,A 0.000,B 0.000,C 90.000,E1 316.986} C_DIS
LIN {X 0.014,Y -234.700,Z 1107.744,A 0.000,B 0.000,C 90.000,E1 313.947} C_DIS
LIN {X 0.110,Y -244.192,Z 1107.730,A 0.000,B 0.000,C 90.000,E1 311.310} C_DIS
LIN {X 0.082,Y -253.296,Z 1107.717,A 0.000,B 0.000,C 90.000,E1 309.116} C_DIS
LIN {X 0.056,Y -266.848,Z 1107.701,A 0.000,B 0.000,C 90.000,E1 306.251} C_DIS
LIN {X 0.177,Y -283.552,Z 1107.684,A 0.000,B 0.000,C 90.000,E1 303.086} C_DIS
LIN {X 0.013,Y -301.640,Z 1107.667,A 0.000,B 0.000,C 90.000,E1 300.079} C_DIS
LIN {X 0.065,Y -321.601,Z 1107.651,A 0.000,B 0.000,C 90.000,E1 297.129} C_DIS
LIN {X 0.176,Y -336.057,Z 1107.640,A 0.000,B 0.000,C 90.000,E1 295.207} C_DIS
LIN {X 0.055,Y -351.692,Z 1107.630,A 0.000,B 0.000,C 90.000,E1 293.387} C_DIS
LIN {X 0.120,Y -364.935,Z 1107.622,A 0.000,B 0.000,C 90.000,E1 291.972} C_DIS
LIN {X -0.048,Y -378.127,Z 1107.615,A 0.000,B 0.000,C 90.000,E1 290.737} C_DIS
LIN {X -0.059,Y -394.709,Z 1107.607,A 0.000,B 0.000,C 90.000,E1 289.268} C_DIS
LIN {X 0.114,Y -408.136,Z 1107.600,A 0.000,B 0.000,C 90.000,E1 288.055} C_DIS
LIN {X 0.075,Y -418.611,Z 1107.595,A 0.000,B 0.000,C 90.000,E1 287.094} C_DIS
LIN {X -0.140,Y -426.278,Z 1107.591,A 0.000,B 0.000,C 90.000,E1 286.386} C_DIS
LIN {X -0.062,Y -433.845,Z 1107.587,A 0.000,B 0.000,C 90.000,E1 285.607} C_DIS
LIN {X -0.121,Y -441.046,Z 1107.582,A 0.000,B 0.000,C 90.000,E1 284.828} C_DIS
LIN {X 0.092,Y -447.782,Z 1107.578,A 0.000,B 0.000,C 90.000,E1 284.008} C_DIS
LIN {X -0.069,Y -453.919,Z 1107.573,A 0.000,B 0.000,C 90.000,E1 283.244} C_DIS
LIN {X -0.172,Y -459.346,Z 1107.569,A 0.000,B 0.000,C 90.000,E1 282.479} C_DIS
LIN {X -0.235,Y -464.045,Z 1107.565,A 0.000,B 0.000,C 90.000,E1 281.715} C_DIS
LIN {X -0.101,Y -466.873,Z 1107.562,A 0.000,B 0.000,C 90.000,E1 281.186} C_DIS
LIN {X -0.099,Y -470.531,Z 1107.558,A 0.000,B 0.000,C 90.000,E1 280.423} C_DIS
LIN {X -0.155,Y -473.588,Z 1107.554,A 0.000,B 0.000,C 90.000,E1 279.670} C_DIS
LIN {X -0.049,Y -475.270,Z 1107.551,A 0.000,B 0.000,C 90.000,E1 279.151} C_DIS
LIN {X 0.145,Y -476.674,Z 1107.548,A 0.000,B 0.000,C 90.000,E1 278.624} C_DIS
LIN {X -0.196,Y -477.839,Z 1107.545,A 0.000,B 0.000,C 90.000,E1 278.163} C_DIS
LIN {X -0.055,Y -478.783,Z 1107.542,A 0.000,B 0.000,C 90.000,E1 277.644} C_DIS
LIN {X 0.094,Y -479.393,Z 1107.540,A 0.000,B 0.000,C 90.000,E1 277.125} C_DIS
LIN {X -0.225,Y -479.783,Z 1107.537,A 0.000,B 0.000,C 90.000,E1 276.663} C_DIS
LIN {X -0.066,Y -479.850,Z 1107.534,A 0.000,B 0.000,C 90.000,E1 276.144} C_DIS
LIN {X 0.096,Y -479.608,Z 1107.531,A 0.000,B 0.000,C 90.000,E1 275.625} C_DIS
LIN {X -0.220,Y -479.035,Z 1107.529,A 0.000,B 0.000,C 90.000,E1 275.163} C_DIS
LIN {X -0.062,Y -478.081,Z 1107.526,A 0.000,B 0.000,C 90.000,E1 274.645} C_DIS
LIN {X 0.055,Y -476.664,Z 1107.523,A 0.000,B 0.000,C 90.000,E1 274.131} C_DIS
LIN {X 0.202,Y -474.727,Z 1107.520,A 0.000,B 0.000,C 90.000,E1 273.612} C_DIS
LIN {X -0.136,Y -472.150,Z 1107.517,A 0.000,B 0.000,C 90.000,E1 273.151} C_DIS
LIN {X 0.144,Y -470.643,Z 1107.516,A 0.000,B 0.000,C 90.000,E1 272.865} C_DIS
LIN {X 0.226,Y -466.771,Z 1107.513,A 0.000,B 0.000,C 90.000,E1 272.350} C_DIS
LIN {X 0.031,Y -464.504,Z 1107.512,A 0.000,B 0.000,C 90.000,E1 272.121} C_DIS
LIN {X -0.172,Y -461.856,Z 1107.510,A 0.000,B 0.000,C 90.000,E1 271.892} C_DIS
LIN {X 0.100,Y -458.885,Z 1107.509,A 0.000,B 0.000,C 90.000,E1 271.604} C_DIS
LIN {X 0.154,Y -452.644,Z 1107.506,A 0.000,B 0.000,C 90.000,E1 271.146} C_DIS
LIN {X -0.026,Y -449.495,Z 1107.505,A 0.000,B 0.000,C 90.000,E1 270.974} C_DIS
LIN {X -0.102,Y -442.622,Z 1107.503,A 0.000,B 0.000,C 90.000,E1 270.630} C_DIS
LIN {X -0.143,Y -435.619,Z 1107.502,A 0.000,B 0.000,C 90.000,E1 270.344} C_DIS
LIN {X 0.198,Y -428.325,Z 1107.500,A 0.000,B 0.000,C 90.000,E1 270.057} C_DIS
LIN {X 0.022,Y -421.115,Z 1107.499,A 0.000,B 0.000,C 90.000,E1 269.885} C_DIS
LIN {X 0.123,Y -413.611,Z 1107.499,A 0.000,B 0.000,C 90.000,E1 269.714} C_DIS
LIN {X 0.035,Y -405.686,Z 1107.498,A 0.000,B 0.000,C 90.000,E1 269.599} C_DIS
LIN {X 0.166,Y -394.801,Z 1107.497,A 0.000,B 0.000,C 90.000,E1 269.484} C_DIS
LIN {X -0.036,Y -384.334,Z 1107.497,A 0.000,B 0.000,C 90.000,E1 269.484} C_DIS
LIN {X -0.048,Y -181.431,Z 1107.497,A 0.000,B 0.000,C 90.000,E1 269.484} C_DIS
LIN {X 0.076,Y -180.841,Z 1107.472,A 0.000,B 0.000,C 90.000,E1 264.894} C_DIS
LIN {X -0.022,Y -178.949,Z 1107.444,A 0.000,B 0.000,C 90.000,E1 259.859} C_DIS
LIN {X -0.005,Y -176.853,Z 1107.425,A 0.000,B 0.000,C 90.000,E1 256.464} C_DIS
LIN {X -0.033,Y -175.512,Z 1107.411,A 0.000,B 0.000,C 90.000,E1 253.921} C_DIS
LIN {X 0.029,Y -172.252,Z 1107.387,A 0.000,B 0.000,C 90.000,E1 249.625} C_DIS
LIN {X 0.007,Y -171.730,Z 1107.382,A 0.000,B 0.000,C 90.000,E1 248.773} C_DIS
LIN {X 0.017,Y -167.327,Z 1107.353,A 0.000,B 0.000,C 90.000,E1 243.589} C_DIS
LIN {X -0.052,Y -166.710,Z 1107.349,A 0.000,B 0.000,C 90.000,E1 242.743} C_DIS
LIN {X 0.086,Y -162.691,Z 1107.324,A 0.000,B 0.000,C 90.000,E1 238.329} C_DIS
LIN {X -0.076,Y -161.381,Z 1107.314,A 0.000,B 0.000,C 90.000,E1 236.628} C_DIS
LIN {X -0.032,Y -157.374,Z 1107.290,A 0.000,B 0.000,C 90.000,E1 232.190} C_DIS
LIN {X 0.002,Y -155.367,Z 1107.275,A 0.000,B 0.000,C 90.000,E1 229.504} C_DIS
LIN {X 0.049,Y -151.708,Z 1107.250,A 0.000,B 0.000,C 90.000,E1 225.000} C_DIS
LIN {X 0.058,Y -149.898,Z 1107.235,A 0.000,B 0.000,C 90.000,E1 222.285} C_DIS
LIN {X 0.082,Y -146.758,Z 1107.210,A 0.000,B 0.000,C 90.000,E1 217.729} C_DIS
LIN {X -0.019,Y -145.325,Z 1107.195,A 0.000,B 0.000,C 90.000,E1 215.025} C_DIS
LIN {X 0.020,Y -142.409,Z 1107.164,A 0.000,B 0.000,C 90.000,E1 209.489} C_DIS
LIN {X -0.053,Y -141.393,Z 1107.148,A 0.000,B 0.000,C 90.000,E1 206.744} C_DIS
LIN {X -0.066,Y -139.352,Z 1107.112,A 0.000,B 0.000,C 90.000,E1 200.248} C_DIS
LIN {X 0.055,Y -138.792,Z 1107.097,A 0.000,B 0.000,C 90.000,E1 197.402} C_DIS
LIN {X -0.022,Y -138.346,Z 1107.055,A 0.000,B 0.000,C 90.000,E1 189.962} C_DIS
LIN {X -0.005,Y -139.380,Z 1107.009,A 0.000,B 0.000,C 90.000,E1 181.547} C_DIS
LIN {X 0.048,Y -141.272,Z 1106.972,A 0.000,B 0.000,C 90.000,E1 175.008} C_DIS
LIN {X 0.006,Y -142.638,Z 1106.957,A 0.000,B 0.000,C 90.000,E1 172.243} C_DIS
LIN {X -0.042,Y -144.967,Z 1106.931,A 0.000,B 0.000,C 90.000,E1 167.645} C_DIS
LIN {X -0.051,Y -147.596,Z 1106.911,A 0.000,B 0.000,C 90.000,E1 163.976} C_DIS
LIN {X -0.022,Y -150.213,Z 1106.891,A 0.000,B 0.000,C 90.000,E1 160.315} C_DIS
LIN {X 0.045,Y -153.599,Z 1106.870,A 0.000,B 0.000,C 90.000,E1 156.666} C_DIS
LIN {X 0.033,Y -157.016,Z 1106.850,A 0.000,B 0.000,C 90.000,E1 153.076} C_DIS
LIN {X -0.035,Y -161.136,Z 1106.831,A 0.000,B 0.000,C 90.000,E1 149.537} C_DIS
LIN {X 0.048,Y -163.235,Z 1106.821,A 0.000,B 0.000,C 90.000,E1 147.740} C_DIS
LIN {X -0.087,Y -167.668,Z 1106.801,A 0.000,B 0.000,C 90.000,E1 144.276} C_DIS
LIN {X 0.062,Y -171.492,Z 1106.787,A 0.000,B 0.000,C 90.000,E1 141.618} C_DIS
LIN {X 0.106,Y -176.424,Z 1106.768,A 0.000,B 0.000,C 90.000,E1 138.162} C_DIS
LIN {X -0.023,Y -180.719,Z 1106.754,A 0.000,B 0.000,C 90.000,E1 135.648} C_DIS
LIN {X -0.042,Y -186.122,Z 1106.735,A 0.000,B 0.000,C 90.000,E1 132.285} C_DIS
LIN {X 0.016,Y -190.760,Z 1106.721,A 0.000,B 0.000,C 90.000,E1 129.769} C_DIS
LIN {X -0.075,Y -196.515,Z 1106.703,A 0.000,B 0.000,C 90.000,E1 126.503} C_DIS
LIN {X -0.031,Y -200.261,Z 1106.692,A 0.000,B 0.000,C 90.000,E1 124.612} C_DIS
LIN {X -0.096,Y -308.769,Z 1106.692,A 0.000,B 0.000,C 90.000,E1 124.612} C_DIS
LIN {X 0.017,Y -313.055,Z 1106.691,A 0.000,B 0.000,C 90.000,E1 124.452} C_DIS
LIN {X -0.047,Y -315.218,Z 1106.691,A 0.000,B 0.000,C 90.000,E1 124.326} C_DIS
LIN {X 0.003,Y -318.179,Z 1106.689,A 0.000,B 0.000,C 90.000,E1 124.040} C_DIS
LIN {X 0.051,Y -321.844,Z 1106.686,A 0.000,B 0.000,C 90.000,E1 123.499} C_DIS
LIN {X 0.127,Y -323.384,Z 1106.684,A 0.000,B 0.000,C 90.000,E1 123.166} C_DIS
LIN {X -0.155,Y -336.446,Z 1106.665,A 0.000,B 0.000,C 90.000,E1 119.745} C_DIS
LIN {X -0.058,Y -348.553,Z 1106.650,A 0.000,B 0.000,C 90.000,E1 116.950} C_DIS
LIN {X 0.073,Y -362.141,Z 1106.635,A 0.000,B 0.000,C 90.000,E1 114.207} C_DIS
LIN {X 0.047,Y -375.553,Z 1106.621,A 0.000,B 0.000,C 90.000,E1 111.844} C_DIS
LIN {X 0.084,Y -390.321,Z 1106.609,A 0.000,B 0.000,C 90.000,E1 109.523} C_DIS
LIN {X -0.017,Y -406.548,Z 1106.596,A 0.000,B 0.000,C 90.000,E1 107.275} C_DIS
LIN {X 0.024,Y -424.351,Z 1106.584,A 0.000,B 0.000,C 90.000,E1 105.064} C_DIS
LIN {X -0.071,Y -443.772,Z 1106.572,A 0.000,B 0.000,C 90.000,E1 102.939} C_DIS
LIN {X -0.024,Y -463.990,Z 1106.561,A 0.000,B 0.000,C 90.000,E1 100.950} C_DIS
LIN {X -0.095,Y -468.986,Z 1106.558,A 0.000,B 0.000,C 90.000,E1 100.489} C_DIS
LIN {X -0.145,Y -470.902,Z 1106.557,A 0.000,B 0.000,C 90.000,E1 100.254} C_DIS
LIN {X -0.196,Y -472.356,Z 1106.556,A 0.000,B 0.000,C 90.000,E1 100.018} C_DIS
LIN {X -0.096,Y -474.329,Z 1106.553,A 0.000,B 0.000,C 90.000,E1 99.500} C_DIS
LIN {X 0.092,Y -475.180,Z 1106.550,A 0.000,B 0.000,C 90.000,E1 98.973} C_DIS
LIN {X 0.216,Y -475.053,Z 1106.547,A 0.000,B 0.000,C 90.000,E1 98.454} C_DIS
LIN {X -0.122,Y -473.938,Z 1106.544,A 0.000,B 0.000,C 90.000,E1 97.992} C_DIS
LIN {X 0.211,Y -472.958,Z 1106.543,A 0.000,B 0.000,C 90.000,E1 97.701} C_DIS
LIN {X 0.072,Y -471.636,Z 1106.542,A 0.000,B 0.000,C 90.000,E1 97.466} C_DIS
LIN {X -0.084,Y -457.235,Z 1106.530,A 0.000,B 0.000,C 90.000,E1 95.454} C_DIS
LIN {X 0.113,Y -441.279,Z 1106.517,A 0.000,B 0.000,C 90.000,E1 93.094} C_DIS
LIN {X 0.117,Y -428.215,Z 1106.505,A 0.000,B 0.000,C 90.000,E1 90.974} C_DIS
LIN {X -0.074,Y -414.284,Z 1106.492,A 0.000,B 0.000,C 90.000,E1 88.568} C_DIS
LIN {X 0.100,Y -403.909,Z 1106.481,A 0.000,B 0.000,C 90.000,E1 86.617} C_DIS
LIN {X 0.114,Y -391.763,Z 1106.469,A 0.000,B 0.000,C 90.000,E1 84.375} C_DIS
LIN {X -0.099,Y -381.191,Z 1106.458,A 0.000,B 0.000,C 90.000,E1 82.413} C_DIS
LIN {X -0.107,Y -371.981,Z 1106.448,A 0.000,B 0.000,C 90.000,E1 80.679} C_DIS
LIN {X 0.197,Y -362.417,Z 1106.438,A 0.000,B 0.000,C 90.000,E1 78.870} C_DIS
LIN {X -0.030,Y -352.544,Z 1106.428,A 0.000,B 0.000,C 90.000,E1 77.117} C_DIS
LIN {X -0.020,Y -339.308,Z 1106.415,A 0.000,B 0.000,C 90.000,E1 74.685} C_DIS
LIN {X 0.043,Y -324.777,Z 1106.399,A 0.000,B 0.000,C 90.000,E1 71.873} C_DIS
LIN {X -0.090,Y -311.046,Z 1106.383,A 0.000,B 0.000,C 90.000,E1 69.028} C_DIS
LIN {X -0.036,Y -299.572,Z 1106.369,A 0.000,B 0.000,C 90.000,E1 66.410} C_DIS
LIN {X -0.139,Y -288.418,Z 1106.354,A 0.000,B 0.000,C 90.000,E1 63.768} C_DIS
LIN {X -0.134,Y -277.621,Z 1106.339,A 0.000,B 0.000,C 90.000,E1 61.051} C_DIS
LIN {X 0.007,Y -267.080,Z 1106.324,A 0.000,B 0.000,C 90.000,E1 58.250} C_DIS
LIN {X 0.046,Y -255.681,Z 1106.306,A 0.000,B 0.000,C 90.000,E1 55.055} C_DIS
LIN {X -0.060,Y -244.911,Z 1106.288,A 0.000,B 0.000,C 90.000,E1 51.823} C_DIS
LIN {X 0.021,Y -235.998,Z 1106.271,A 0.000,B 0.000,C 90.000,E1 48.852} C_DIS
LIN {X -0.140,Y -227.708,Z 1106.255,A 0.000,B 0.000,C 90.000,E1 45.891} C_DIS
LIN {X -0.028,Y -219.789,Z 1106.238,A 0.000,B 0.000,C 90.000,E1 42.813} C_DIS
LIN {X -0.076,Y -212.271,Z 1106.221,A 0.000,B 0.000,C 90.000,E1 39.725} C_DIS
LIN {X -0.108,Y -205.180,Z 1106.203,A 0.000,B 0.000,C 90.000,E1 36.583} C_DIS
LIN {X -0.064,Y -198.579,Z 1106.185,A 0.000,B 0.000,C 90.000,E1 33.372} C_DIS
LIN {X -0.069,Y -192.606,Z 1106.167,A 0.000,B 0.000,C 90.000,E1 30.129} C_DIS
LIN {X -0.006,Y -187.201,Z 1106.149,A 0.000,B 0.000,C 90.000,E1 26.821} C_DIS
LIN {X -0.073,Y -182.557,Z 1106.130,A 0.000,B 0.000,C 90.000,E1 23.515} C_DIS
LIN {X 0.026,Y -178.567,Z 1106.112,A 0.000,B 0.000,C 90.000,E1 20.120} C_DIS
LIN {X -0.047,Y -174.533,Z 1106.088,A 0.000,B 0.000,C 90.000,E1 15.898} C_DIS
LIN {X 0.024,Y -171.562,Z 1106.064,A 0.000,B 0.000,C 90.000,E1 11.591} C_DIS
LIN {X -0.032,Y -169.124,Z 1106.031,A 0.000,B 0.000,C 90.000,E1 5.568} C_DIS
LIN {X 0.021,Y -170.318,Z 1105.959,A 0.000,B 0.000,C 90.000,E1 352.591} C_DIS
LIN {X 0.038,Y -173.206,Z 1105.930,A 0.000,B 0.000,C 90.000,E1 347.409} C_DIS
LIN {X -0.013,Y -176.708,Z 1105.906,A 0.000,B 0.000,C 90.000,E1 343.142} C_DIS
LIN {X -0.034,Y -181.169,Z 1105.883,A 0.000,B 0.000,C 90.000,E1 338.901} C_DIS
LIN {X -0.041,Y -185.535,Z 1105.864,A 0.000,B 0.000,C 90.000,E1 335.537} C_DIS
LIN {X -0.126,Y -190.580,Z 1105.845,A 0.000,B 0.000,C 90.000,E1 332.231} C_DIS
LIN {X 0.104,Y -196.436,Z 1105.827,A 0.000,B 0.000,C 90.000,E1 328.869} C_DIS
LIN {X -0.087,Y -202.921,Z 1105.809,A 0.000,B 0.000,C 90.000,E1 325.674} C_DIS
LIN {X -0.111,Y -210.164,Z 1105.791,A 0.000,B 0.000,C 90.000,E1 322.477} C_DIS
LIN {X -0.092,Y -219.253,Z 1105.772,A 0.000,B 0.000,C 90.000,E1 318.933} C_DIS
LIN {X 0.056,Y -228.336,Z 1105.755,A 0.000,B 0.000,C 90.000,E1 315.810} C_DIS
LIN {X 0.119,Y -238.459,Z 1105.738,A 0.000,B 0.000,C 90.000,E1 312.771} C_DIS
LIN {X -0.050,Y -248.482,Z 1105.723,A 0.000,B 0.000,C 90.000,E1 310.216} C_DIS
LIN {X -0.057,Y -261.542,Z 1105.707,A 0.000,B 0.000,C 90.000,E1 307.317} C_DIS
LIN {X -0.027,Y -275.903,Z 1105.692,A 0.000,B 0.000,C 90.000,E1 304.485} C_DIS
LIN {X 0.042,Y -293.384,Z 1105.674,A 0.000,B 0.000,C 90.000,E1 301.386} C_DIS
LIN {X -0.041,Y -310.318,Z 1105.660,A 0.000,B 0.000,C 90.000,E1 298.743} C_DIS
LIN {X -0.042,Y -331.197,Z 1105.644,A 0.000,B 0.000,C 90.000,E1 295.848} C_DIS
LIN {X -0.097,Y -346.326,Z 1105.633,A 0.000,B 0.000,C 90.000,E1 294.003} C_DIS
LIN {X -0.021,Y -359.721,Z 1105.625,A 0.000,B 0.000,C 90.000,E1 292.514} C_DIS
LIN {X -0.062,Y -376.014,Z 1105.616,A 0.000,B 0.000,C 90.000,E1 290.918} C_DIS
LIN {X -0.059,Y -395.214,Z 1105.607,A 0.000,B 0.000,C 90.000,E1 289.214} C_DIS
LIN {X 0.084,Y -408.691,Z 1105.600,A 0.000,B 0.000,C 90.000,E1 288.000} C_DIS
LIN {X 0.011,Y -419.261,Z 1105.595,A 0.000,B 0.000,C 90.000,E1 287.040} C_DIS
LIN {X -0.125,Y -426.975,Z 1105.591,A 0.000,B 0.000,C 90.000,E1 286.315} C_DIS
LIN {X 0.182,Y -436.963,Z 1105.585,A 0.000,B 0.000,C 90.000,E1 285.245} C_DIS
LIN {X -0.041,Y -444.015,Z 1105.580,A 0.000,B 0.000,C 90.000,E1 284.481} C_DIS
LIN {X -0.132,Y -450.545,Z 1105.576,A 0.000,B 0.000,C 90.000,E1 283.703} C_DIS
LIN {X 0.174,Y -456.346,Z 1105.572,A 0.000,B 0.000,C 90.000,E1 282.883} C_DIS
LIN {X 0.086,Y -461.522,Z 1105.567,A 0.000,B 0.000,C 90.000,E1 282.119} C_DIS
LIN {X -0.048,Y -466.015,Z 1105.563,A 0.000,B 0.000,C 90.000,E1 281.366} C_DIS
LIN {X -0.054,Y -469.850,Z 1105.559,A 0.000,B 0.000,C 90.000,E1 280.602} C_DIS
LIN {X 0.113,Y -472.026,Z 1105.556,A 0.000,B 0.000,C 90.000,E1 280.074} C_DIS
LIN {X 0.215,Y -473.961,Z 1105.553,A 0.000,B 0.000,C 90.000,E1 279.557} C_DIS
LIN {X -0.144,Y -475.623,Z 1105.550,A 0.000,B 0.000,C 90.000,E1 279.095} C_DIS
LIN {X 0.053,Y -476.982,Z 1105.548,A 0.000,B 0.000,C 90.000,E1 278.568} C_DIS
LIN {X 0.187,Y -478.135,Z 1105.545,A 0.000,B 0.000,C 90.000,E1 278.049} C_DIS
LIN {X -0.143,Y -479.043,Z 1105.542,A 0.000,B 0.000,C 90.000,E1 277.587} C_DIS
LIN {X 0.010,Y -479.672,Z 1105.539,A 0.000,B 0.000,C 90.000,E1 277.068} C_DIS
LIN {X 0.168,Y -480.026,Z 1105.536,A 0.000,B 0.000,C 90.000,E1 276.549} C_DIS
LIN {X -0.147,Y -480.087,Z 1105.534,A 0.000,B 0.000,C 90.000,E1 276.087} C_DIS
LIN {X 0.017,Y -479.821,Z 1105.531,A 0.000,B 0.000,C 90.000,E1 275.568} C_DIS
LIN {X 0.180,Y -479.199,Z 1105.528,A 0.000,B 0.000,C 90.000,E1 275.049} C_DIS
LIN {X -0.138,Y -478.186,Z 1105.525,A 0.000,B 0.000,C 90.000,E1 274.588} C_DIS
LIN {X -0.019,Y -476.738,Z 1105.523,A 0.000,B 0.000,C 90.000,E1 274.073} C_DIS
LIN {X 0.129,Y -474.764,Z 1105.520,A 0.000,B 0.000,C 90.000,E1 273.555} C_DIS
LIN {X -0.209,Y -472.138,Z 1105.517,A 0.000,B 0.000,C 90.000,E1 273.094} C_DIS
LIN {X -0.117,Y -468.719,Z 1105.514,A 0.000,B 0.000,C 90.000,E1 272.579} C_DIS
LIN {X -0.040,Y -464.254,Z 1105.511,A 0.000,B 0.000,C 90.000,E1 272.064} C_DIS
LIN {X 0.233,Y -461.592,Z 1105.510,A 0.000,B 0.000,C 90.000,E1 271.776} C_DIS
LIN {X 0.078,Y -455.589,Z 1105.507,A 0.000,B 0.000,C 90.000,E1 271.318} C_DIS
LIN {X -0.017,Y -449.121,Z 1105.505,A 0.000,B 0.000,C 90.000,E1 270.917} C_DIS
LIN {X -0.051,Y -442.311,Z 1105.503,A 0.000,B 0.000,C 90.000,E1 270.573} C_DIS
LIN {X -0.065,Y -435.215,Z 1105.502,A 0.000,B 0.000,C 90.000,E1 270.286} C_DIS
LIN {X -0.114,Y -427.970,Z 1105.500,A 0.000,B 0.000,C 90.000,E1 270.057} C_DIS
LIN {X 0.177,Y -420.550,Z 1105.499,A 0.000,B 0.000,C 90.000,E1 269.828} C_DIS
LIN {X -0.104,Y -413.137,Z 1105.498,A 0.000,B 0.000,C 90.000,E1 269.714} C_DIS
LIN {X -0.152,Y -404.907,Z 1105.498,A 0.000,B 0.000,C 90.000,E1 269.599} C_DIS
LIN {X 0.139,Y -397.101,Z 1105.497,A 0.000,B 0.000,C 90.000,E1 269.484} C_DIS
LIN {X -0.069,Y -389.801,Z 1105.497,A 0.000,B 0.000,C 90.000,E1 269.484} C_DIS
LIN {X -0.064,Y -181.430,Z 1105.497,A 0.000,B 0.000,C 90.000,E1 269.484} C_DIS
LIN {X -0.027,Y -180.899,Z 1105.474,A 0.000,B 0.000,C 90.000,E1 265.241} C_DIS
LIN {X -0.077,Y -180.214,Z 1105.464,A 0.000,B 0.000,C 90.000,E1 263.571} C_DIS
LIN {X 0.053,Y -179.033,Z 1105.445,A 0.000,B 0.000,C 90.000,E1 260.151} C_DIS
LIN {X -0.061,Y -178.690,Z 1105.441,A 0.000,B 0.000,C 90.000,E1 259.342} C_DIS
LIN {X 0.050,Y -175.739,Z 1105.412,A 0.000,B 0.000,C 90.000,E1 254.212} C_DIS
LIN {X 0.046,Y -171.923,Z 1105.384,A 0.000,B 0.000,C 90.000,E1 249.082} C_DIS
LIN {X 0.020,Y -171.296,Z 1105.379,A 0.000,B 0.000,C 90.000,E1 248.230} C_DIS
LIN {X 0.065,Y -167.559,Z 1105.355,A 0.000,B 0.000,C 90.000,E1 243.896} C_DIS
LIN {X 0.079,Y -166.183,Z 1105.345,A 0.000,B 0.000,C 90.000,E1 242.153} C_DIS
LIN {X 0.068,Y -162.953,Z 1105.326,A 0.000,B 0.000,C 90.000,E1 238.663} C_DIS
LIN {X -0.108,Y -160.861,Z 1105.311,A 0.000,B 0.000,C 90.000,E1 236.087} C_DIS
LIN {X 0.093,Y -157.636,Z 1105.292,A 0.000,B 0.000,C 90.000,E1 232.477} C_DIS
LIN {X 0.031,Y -155.674,Z 1105.277,A 0.000,B 0.000,C 90.000,E1 229.828} C_DIS
LIN {X 0.082,Y -151.940,Z 1105.252,A 0.000,B 0.000,C 90.000,E1 225.324} C_DIS
LIN {X 0.097,Y -150.178,Z 1105.237,A 0.000,B 0.000,C 90.000,E1 222.609} C_DIS
LIN {X 0.017,Y -146.954,Z 1105.212,A 0.000,B 0.000,C 90.000,E1 218.096} C_DIS
LIN {X 0.004,Y -145.541,Z 1105.196,A 0.000,B 0.000,C 90.000,E1 215.358} C_DIS
LIN {X -0.080,Y -142.937,Z 1105.171,A 0.000,B 0.000,C 90.000,E1 210.797} C_DIS
LIN {X -0.022,Y -141.561,Z 1105.150,A 0.000,B 0.000,C 90.000,E1 207.078} C_DIS
LIN {X 0.030,Y -139.409,Z 1105.114,A 0.000,B 0.000,C 90.000,E1 200.556} C_DIS
LIN {X -0.048,Y -139.130,Z 1105.104,A 0.000,B 0.000,C 90.000,E1 198.725} C_DIS
LIN {X -0.020,Y -138.350,Z 1105.057,A 0.000,B 0.000,C 90.000,E1 190.310} C_DIS
LIN {X -0.033,Y -139.498,Z 1105.005,A 0.000,B 0.000,C 90.000,E1 180.974} C_DIS
LIN {X 0.048,Y -141.120,Z 1104.974,A 0.000,B 0.000,C 90.000,E1 175.355} C_DIS
LIN {X 0.001,Y -142.500,Z 1104.959,A 0.000,B 0.000,C 90.000,E1 172.591} C_DIS
LIN {X -0.052,Y -144.755,Z 1104.933,A 0.000,B 0.000,C 90.000,E1 167.993} C_DIS
LIN {X 0.039,Y -147.364,Z 1104.913,A 0.000,B 0.000,C 90.000,E1 164.283} C_DIS
LIN {X -0.039,Y -150.691,Z 1104.887,A 0.000,B 0.000,C 90.000,E1 159.752} C_DIS
LIN {X 0.044,Y -154.171,Z 1104.867,A 0.000,B 0.000,C 90.000,E1 156.102} C_DIS
LIN {X -0.026,Y -157.606,Z 1104.847,A 0.000,B 0.000,C 90.000,E1 152.538} C_DIS
LIN {X -0.075,Y -161.858,Z 1104.828,A 0.000,B 0.000,C 90.000,E1 148.997} C_DIS
LIN {X -0.058,Y -166.048,Z 1104.808,A 0.000,B 0.000,C 90.000,E1 145.468} C_DIS
LIN {X -0.067,Y -171.052,Z 1104.789,A 0.000,B 0.000,C 90.000,E1 141.984} C_DIS
LIN {X -0.038,Y -175.924,Z 1104.770,A 0.000,B 0.000,C 90.000,E1 138.528} C_DIS
LIN {X -0.045,Y -180.163,Z 1104.755,A 0.000,B 0.000,C 90.000,E1 135.972} C_DIS
LIN {X -0.076,Y -185.580,Z 1104.737,A 0.000,B 0.000,C 90.000,E1 132.609} C_DIS
LIN {X -0.026,Y -190.170,Z 1104.723,A 0.000,B 0.000,C 90.000,E1 130.092} C_DIS
LIN {X 0.018,Y -197.499,Z 1104.700,A 0.000,B 0.000,C 90.000,E1 125.964} C_DIS
LIN {X 0.062,Y -200.205,Z 1104.692,A 0.000,B 0.000,C 90.000,E1 124.612} C_DIS
LIN {X 0.049,Y -308.311,Z 1104.692,A 0.000,B 0.000,C 90.000,E1 124.612} C_DIS
LIN {X -0.046,Y -309.512,Z 1104.692,A 0.000,B 0.000,C 90.000,E1 124.612} C_DIS
LIN {X 0.095,Y -315.080,Z 1104.691,A 0.000,B 0.000,C 90.000,E1 124.326} C_DIS
LIN {X 0.073,Y -318.169,Z 1104.689,A 0.000,B 0.000,C 90.000,E1 124.040} C_DIS
LIN {X 0.111,Y -321.809,Z 1104.686,A 0.000,B 0.000,C 90.000,E1 123.499} C_DIS
LIN {X -0.083,Y -323.335,Z 1104.684,A 0.000,B 0.000,C 90.000,E1 123.214} C_DIS
LIN {X -0.095,Y -336.383,Z 1104.665,A 0.000,B 0.000,C 90.000,E1 119.745} C_DIS
LIN {X 0.003,Y -348.484,Z 1104.650,A 0.000,B 0.000,C 90.000,E1 116.950} C_DIS
LIN {X 0.135,Y -362.065,Z 1104.635,A 0.000,B 0.000,C 90.000,E1 114.207} C_DIS
LIN {X 0.108,Y -375.473,Z 1104.621,A 0.000,B 0.000,C 90.000,E1 111.844} C_DIS
LIN {X -0.222,Y -390.234,Z 1104.609,A 0.000,B 0.000,C 90.000,E1 109.577} C_DIS
LIN {X 0.045,Y -406.455,Z 1104.596,A 0.000,B 0.000,C 90.000,E1 107.275} C_DIS
LIN {X 0.087,Y -424.251,Z 1104.584,A 0.000,B 0.000,C 90.000,E1 105.064} C_DIS
LIN {X -0.010,Y -443.668,Z 1104.572,A 0.000,B 0.000,C 90.000,E1 102.939} C_DIS
LIN {X 0.033,Y -463.885,Z 1104.561,A 0.000,B 0.000,C 90.000,E1 100.950} C_DIS
LIN {X -0.038,Y -468.894,Z 1104.558,A 0.000,B 0.000,C 90.000,E1 100.489} C_DIS
LIN {X -0.082,Y -470.821,Z 1104.557,A 0.000,B 0.000,C 90.000,E1 100.254} C_DIS
LIN {X -0.128,Y -472.284,Z 1104.556,A 0.000,B 0.000,C 90.000,E1 100.018} C_DIS
LIN {X -0.027,Y -474.280,Z 1104.553,A 0.000,B 0.000,C 90.000,E1 99.500} C_DIS
LIN {X 0.161,Y -475.147,Z 1104.550,A 0.000,B 0.000,C 90.000,E1 98.973} C_DIS
LIN {X -0.185,Y -475.038,Z 1104.547,A 0.000,B 0.000,C 90.000,E1 98.511} C_DIS
LIN {X -0.053,Y -473.940,Z 1104.544,A 0.000,B 0.000,C 90.000,E1 97.992} C_DIS
LIN {X -0.190,Y -472.972,Z 1104.543,A 0.000,B 0.000,C 90.000,E1 97.757} C_DIS
LIN {X 0.078,Y -471.663,Z 1104.542,A 0.000,B 0.000,C 90.000,E1 97.473} C_DIS
LIN {X -0.017,Y -457.262,Z 1104.530,A 0.000,B 0.000,C 90.000,E1 95.454} C_DIS
LIN {X 0.179,Y -441.298,Z 1104.517,A 0.000,B 0.000,C 90.000,E1 93.094} C_DIS
LIN {X 0.182,Y -428.242,Z 1104.505,A 0.000,B 0.000,C 90.000,E1 90.974} C_DIS
LIN {X -0.011,Y -414.302,Z 1104.492,A 0.000,B 0.000,C 90.000,E1 88.568} C_DIS
LIN {X 0.163,Y -403.935,Z 1104.481,A 0.000,B 0.000,C 90.000,E1 86.617} C_DIS
LIN {X 0.120,Y -393.320,Z 1104.470,A 0.000,B 0.000,C 90.000,E1 84.666} C_DIS
LIN {X -0.039,Y -381.201,Z 1104.458,A 0.000,B 0.000,C 90.000,E1 82.413} C_DIS
LIN {X -0.048,Y -371.967,Z 1104.448,A 0.000,B 0.000,C 90.000,E1 80.679} C_DIS
LIN {X -0.102,Y -362.386,Z 1104.438,A 0.000,B 0.000,C 90.000,E1 78.926} C_DIS
LIN {X 0.025,Y -352.512,Z 1104.428,A 0.000,B 0.000,C 90.000,E1 77.117} C_DIS
LIN {X 0.031,Y -340.925,Z 1104.417,A 0.000,B 0.000,C 90.000,E1 74.991} C_DIS
LIN {X 0.133,Y -326.328,Z 1104.401,A 0.000,B 0.000,C 90.000,E1 72.181} C_DIS
LIN {X -0.044,Y -311.024,Z 1104.383,A 0.000,B 0.000,C 90.000,E1 69.028} C_DIS
LIN {X 0.008,Y -299.546,Z 1104.369,A 0.000,B 0.000,C 90.000,E1 66.410} C_DIS
LIN {X -0.097,Y -288.388,Z 1104.354,A 0.000,B 0.000,C 90.000,E1 63.768} C_DIS
LIN {X -0.095,Y -277.572,Z 1104.339,A 0.000,B 0.000,C 90.000,E1 61.051} C_DIS
LIN {X 0.043,Y -267.008,Z 1104.324,A 0.000,B 0.000,C 90.000,E1 58.250} C_DIS
LIN {X 0.078,Y -255.589,Z 1104.306,A 0.000,B 0.000,C 90.000,E1 55.055} C_DIS
LIN {X -0.031,Y -244.787,Z 1104.288,A 0.000,B 0.000,C 90.000,E1 51.823} C_DIS
LIN {X 0.045,Y -235.851,Z 1104.271,A 0.000,B 0.000,C 90.000,E1 48.852} C_DIS
LIN {X -0.121,Y -227.537,Z 1104.255,A 0.000,B 0.000,C 90.000,E1 45.891} C_DIS
LIN {X -0.014,Y -219.605,Z 1104.238,A 0.000,B 0.000,C 90.000,E1 42.813} C_DIS
LIN {X -0.066,Y -212.068,Z 1104.221,A 0.000,B 0.000,C 90.000,E1 39.725} C_DIS
LIN {X -0.104,Y -204.948,Z 1104.203,A 0.000,B 0.000,C 90.000,E1 36.583} C_DIS
LIN {X -0.065,Y -198.326,Z 1104.185,A 0.000,B 0.000,C 90.000,E1 33.372} C_DIS
LIN {X -0.076,Y -192.336,Z 1104.167,A 0.000,B 0.000,C 90.000,E1 30.129} C_DIS
LIN {X -0.020,Y -186.917,Z 1104.149,A 0.000,B 0.000,C 90.000,E1 26.821} C_DIS
LIN {X -0.093,Y -182.288,Z 1104.130,A 0.000,B 0.000,C 90.000,E1 23.515} C_DIS
LIN {X -0.001,Y -178.303,Z 1104.112,A 0.000,B 0.000,C 90.000,E1 20.120} C_DIS
LIN {X 0.086,Y -174.272,Z 1104.088,A 0.000,B 0.000,C 90.000,E1 15.843} C_DIS
LIN {X -0.016,Y -171.316,Z 1104.064,A 0.000,B 0.000,C 90.000,E1 11.591} C_DIS
LIN {X -0.082,Y -168.887,Z 1104.031,A 0.000,B 0.000,C 90.000,E1 5.568} C_DIS
LIN {X 0.008,Y -170.048,Z 1103.959,A 0.000,B 0.000,C 90.000,E1 352.591} C_DIS
LIN {X 0.016,Y -172.923,Z 1103.930,A 0.000,B 0.000,C 90.000,E1 347.409} C_DIS
LIN {X -0.044,Y -176.429,Z 1103.906,A 0.000,B 0.000,C 90.000,E1 343.142} C_DIS
LIN {X -0.075,Y -180.904,Z 1103.883,A 0.000,B 0.000,C 90.000,E1 338.901} C_DIS
LIN {X 0.078,Y -185.269,Z 1103.864,A 0.000,B 0.000,C 90.000,E1 335.485} C_DIS
LIN {X 0.073,Y -190.338,Z 1103.845,A 0.000,B 0.000,C 90.000,E1 332.153} C_DIS
LIN {X 0.039,Y -196.209,Z 1103.827,A 0.000,B 0.000,C 90.000,E1 328.869} C_DIS
LIN {X 0.122,Y -202.705,Z 1103.809,A 0.000,B 0.000,C 90.000,E1 325.595} C_DIS
LIN {X -0.025,Y -209.984,Z 1103.791,A 0.000,B 0.000,C 90.000,E1 322.431} C_DIS
LIN {X 0.127,Y -219.094,Z 1103.772,A 0.000,B 0.000,C 90.000,E1 318.852} C_DIS
LIN {X -0.041,Y -228.172,Z 1103.754,A 0.000,B 0.000,C 90.000,E1 315.810} C_DIS
LIN {X 0.013,Y -238.302,Z 1103.738,A 0.000,B 0.000,C 90.000,E1 312.771} C_DIS
LIN {X 0.026,Y -248.369,Z 1103.723,A 0.000,B 0.000,C 90.000,E1 310.172} C_DIS
LIN {X -0.020,Y -261.458,Z 1103.707,A 0.000,B 0.000,C 90.000,E1 307.282} C_DIS
LIN {X -0.002,Y -275.837,Z 1103.691,A 0.000,B 0.000,C 90.000,E1 304.452} C_DIS
LIN {X -0.080,Y -291.396,Z 1103.676,A 0.000,B 0.000,C 90.000,E1 301.720} C_DIS
LIN {X 0.047,Y -308.146,Z 1103.661,A 0.000,B 0.000,C 90.000,E1 299.027} C_DIS
LIN {X 0.152,Y -328.830,Z 1103.645,A 0.000,B 0.000,C 90.000,E1 296.104} C_DIS
LIN {X 0.034,Y -343.800,Z 1103.635,A 0.000,B 0.000,C 90.000,E1 294.259} C_DIS
LIN {X 0.066,Y -359.455,Z 1103.625,A 0.000,B 0.000,C 90.000,E1 292.514} C_DIS
LIN {X 0.089,Y -375.609,Z 1103.616,A 0.000,B 0.000,C 90.000,E1 290.918} C_DIS
LIN {X -0.091,Y -394.541,Z 1103.607,A 0.000,B 0.000,C 90.000,E1 289.268} C_DIS
LIN {X 0.039,Y -408.090,Z 1103.600,A 0.000,B 0.000,C 90.000,E1 288.055} C_DIS
LIN {X -0.009,Y -418.646,Z 1103.595,A 0.000,B 0.000,C 90.000,E1 287.094} C_DIS
LIN {X -0.094,Y -426.372,Z 1103.591,A 0.000,B 0.000,C 90.000,E1 286.370} C_DIS
LIN {X 0.152,Y -436.377,Z 1103.585,A 0.000,B 0.000,C 90.000,E1 285.315} C_DIS
LIN {X 0.081,Y -443.409,Z 1103.581,A 0.000,B 0.000,C 90.000,E1 284.537} C_DIS
LIN {X -0.120,Y -450.022,Z 1103.576,A 0.000,B 0.000,C 90.000,E1 283.772} C_DIS
LIN {X -0.260,Y -455.916,Z 1103.572,A 0.000,B 0.000,C 90.000,E1 283.008} C_DIS
LIN {X 0.098,Y -461.177,Z 1103.568,A 0.000,B 0.000,C 90.000,E1 282.187} C_DIS
LIN {X 0.058,Y -465.758,Z 1103.563,A 0.000,B 0.000,C 90.000,E1 281.422} C_DIS
LIN {X 0.050,Y -469.662,Z 1103.559,A 0.000,B 0.000,C 90.000,E1 280.658} C_DIS
LIN {X 0.133,Y -471.879,Z 1103.556,A 0.000,B 0.000,C 90.000,E1 280.141} C_DIS
LIN {X -0.152,Y -473.859,Z 1103.554,A 0.000,B 0.000,C 90.000,E1 279.670} C_DIS
LIN {X -0.044,Y -475.549,Z 1103.551,A 0.000,B 0.000,C 90.000,E1 279.151} C_DIS
LIN {X 0.152,Y -476.953,Z 1103.548,A 0.000,B 0.000,C 90.000,E1 278.624} C_DIS
LIN {X -0.189,Y -478.125,Z 1103.545,A 0.000,B 0.000,C 90.000,E1 278.163} C_DIS
LIN {X -0.046,Y -479.070,Z 1103.542,A 0.000,B 0.000,C 90.000,E1 277.644} C_DIS
LIN {X 0.107,Y -479.755,Z 1103.540,A 0.000,B 0.000,C 90.000,E1 277.125} C_DIS
LIN {X -0.213,Y -480.185,Z 1103.537,A 0.000,B 0.000,C 90.000,E1 276.663} C_DIS
LIN {X -0.050,Y -480.266,Z 1103.534,A 0.000,B 0.000,C 90.000,E1 276.144} C_DIS
LIN {X 0.114,Y -480.099,Z 1103.531,A 0.000,B 0.000,C 90.000,E1 275.625} C_DIS
LIN {X -0.200,Y -479.578,Z 1103.529,A 0.000,B 0.000,C 90.000,E1 275.163} C_DIS
LIN {X -0.039,Y -478.645,Z 1103.526,A 0.000,B 0.000,C 90.000,E1 274.645} C_DIS
LIN {X 0.081,Y -477.304,Z 1103.523,A 0.000,B 0.000,C 90.000,E1 274.131} C_DIS
LIN {X 0.230,Y -475.391,Z 1103.520,A 0.000,B 0.000,C 90.000,E1 273.612} C_DIS
LIN {X -0.104,Y -472.892,Z 1103.517,A 0.000,B 0.000,C 90.000,E1 273.151} C_DIS
LIN {X -0.010,Y -469.611,Z 1103.515,A 0.000,B 0.000,C 90.000,E1 272.636} C_DIS
LIN {X 0.070,Y -465.382,Z 1103.512,A 0.000,B 0.000,C 90.000,E1 272.121} C_DIS
LIN {X -0.131,Y -462.842,Z 1103.510,A 0.000,B 0.000,C 90.000,E1 271.892} C_DIS
LIN {X 0.168,Y -457.056,Z 1103.508,A 0.000,B 0.000,C 90.000,E1 271.375} C_DIS
LIN {X 0.191,Y -453.872,Z 1103.506,A 0.000,B 0.000,C 90.000,E1 271.146} C_DIS
LIN {X -0.216,Y -447.209,Z 1103.504,A 0.000,B 0.000,C 90.000,E1 270.802} C_DIS
LIN {X -0.126,Y -440.250,Z 1103.502,A 0.000,B 0.000,C 90.000,E1 270.458} C_DIS
LIN {X -0.029,Y -432.955,Z 1103.501,A 0.000,B 0.000,C 90.000,E1 270.172} C_DIS
LIN {X 0.069,Y -425.713,Z 1103.500,A 0.000,B 0.000,C 90.000,E1 269.943} C_DIS
LIN {X 0.054,Y -418.410,Z 1103.499,A 0.000,B 0.000,C 90.000,E1 269.771} C_DIS
LIN {X -0.144,Y -410.492,Z 1103.498,A 0.000,B 0.000,C 90.000,E1 269.656} C_DIS
LIN {X -0.120,Y -401.646,Z 1103.497,A 0.000,B 0.000,C 90.000,E1 269.542} C_DIS
LIN {X -0.162,Y -390.499,Z 1103.497,A 0.000,B 0.000,C 90.000,E1 269.484} C_DIS
LIN {X 0.072,Y -181.426,Z 1103.497,A 0.000,B 0.000,C 90.000,E1 269.427} C_DIS
LIN {X 0.010,Y -180.836,Z 1103.472,A 0.000,B 0.000,C 90.000,E1 264.894} C_DIS
LIN {X 0.090,Y -178.942,Z 1103.443,A 0.000,B 0.000,C 90.000,E1 259.803} C_DIS
LIN {X -0.044,Y -175.993,Z 1103.415,A 0.000,B 0.000,C 90.000,E1 254.755} C_DIS
LIN {X -0.098,Y -175.495,Z 1103.411,A 0.000,B 0.000,C 90.000,E1 253.921} C_DIS
LIN {X -0.034,Y -172.238,Z 1103.387,A 0.000,B 0.000,C 90.000,E1 249.625} C_DIS
LIN {X -0.055,Y -171.716,Z 1103.382,A 0.000,B 0.000,C 90.000,E1 248.773} C_DIS
LIN {X -0.045,Y -167.312,Z 1103.353,A 0.000,B 0.000,C 90.000,E1 243.589} C_DIS
LIN {X 0.034,Y -166.692,Z 1103.348,A 0.000,B 0.000,C 90.000,E1 242.692} C_DIS
LIN {X 0.026,Y -162.674,Z 1103.324,A 0.000,B 0.000,C 90.000,E1 238.329} C_DIS
LIN {X -0.002,Y -161.364,Z 1103.314,A 0.000,B 0.000,C 90.000,E1 236.580} C_DIS
LIN {X 0.032,Y -157.357,Z 1103.290,A 0.000,B 0.000,C 90.000,E1 232.145} C_DIS
LIN {X 0.061,Y -155.345,Z 1103.275,A 0.000,B 0.000,C 90.000,E1 229.461} C_DIS
LIN {X -0.009,Y -151.692,Z 1103.250,A 0.000,B 0.000,C 90.000,E1 225.000} C_DIS
LIN {X 0.038,Y -150.555,Z 1103.240,A 0.000,B 0.000,C 90.000,E1 223.176} C_DIS
LIN {X -0.045,Y -147.281,Z 1103.215,A 0.000,B 0.000,C 90.000,E1 218.669} C_DIS
LIN {X -0.076,Y -145.310,Z 1103.194,A 0.000,B 0.000,C 90.000,E1 215.025} C_DIS
LIN {X 0.034,Y -142.400,Z 1103.164,A 0.000,B 0.000,C 90.000,E1 209.461} C_DIS
LIN {X 0.017,Y -141.382,Z 1103.148,A 0.000,B 0.000,C 90.000,E1 206.693} C_DIS
LIN {X 0.058,Y -139.349,Z 1103.112,A 0.000,B 0.000,C 90.000,E1 200.174} C_DIS
LIN {X 0.000,Y -138.786,Z 1103.097,A 0.000,B 0.000,C 90.000,E1 197.402} C_DIS
LIN {X 0.058,Y -138.344,Z 1103.055,A 0.000,B 0.000,C 90.000,E1 189.905} C_DIS
LIN {X -0.060,Y -139.386,Z 1103.008,A 0.000,B 0.000,C 90.000,E1 181.547} C_DIS
LIN {X -0.008,Y -141.283,Z 1102.972,A 0.000,B 0.000,C 90.000,E1 175.008} C_DIS
LIN {X -0.050,Y -142.646,Z 1102.957,A 0.000,B 0.000,C 90.000,E1 172.243} C_DIS
LIN {X 0.042,Y -144.982,Z 1102.931,A 0.000,B 0.000,C 90.000,E1 167.589} C_DIS
LIN {X 0.033,Y -147.609,Z 1102.911,A 0.000,B 0.000,C 90.000,E1 163.921} C_DIS
LIN {X -0.030,Y -150.231,Z 1102.891,A 0.000,B 0.000,C 90.000,E1 160.296} C_DIS
LIN {X -0.015,Y -153.622,Z 1102.870,A 0.000,B 0.000,C 90.000,E1 156.666} C_DIS
LIN {X -0.027,Y -157.038,Z 1102.850,A 0.000,B 0.000,C 90.000,E1 153.076} C_DIS
LIN {X -0.096,Y -161.164,Z 1102.831,A 0.000,B 0.000,C 90.000,E1 149.537} C_DIS
LIN {X -0.014,Y -163.259,Z 1102.821,A 0.000,B 0.000,C 90.000,E1 147.740} C_DIS
LIN {X 0.085,Y -167.698,Z 1102.801,A 0.000,B 0.000,C 90.000,E1 144.196} C_DIS
LIN {X -0.002,Y -171.519,Z 1102.787,A 0.000,B 0.000,C 90.000,E1 141.618} C_DIS
LIN {X 0.041,Y -176.456,Z 1102.768,A 0.000,B 0.000,C 90.000,E1 138.162} C_DIS
LIN {X -0.088,Y -180.753,Z 1102.753,A 0.000,B 0.000,C 90.000,E1 135.648} C_DIS
LIN {X 0.030,Y -186.158,Z 1102.735,A 0.000,B 0.000,C 90.000,E1 132.243} C_DIS
LIN {X 0.095,Y -190.796,Z 1102.721,A 0.000,B 0.000,C 90.000,E1 129.725} C_DIS
LIN {X 0.014,Y -196.552,Z 1102.703,A 0.000,B 0.000,C 90.000,E1 126.457} C_DIS
LIN {X -0.045,Y -200.170,Z 1102.693,A 0.000,B 0.000,C 90.000,E1 124.659} C_DIS
LIN {X 0.135,Y -308.575,Z 1102.692,A 0.000,B 0.000,C 90.000,E1 124.612} C_DIS
LIN {X -0.012,Y -313.165,Z 1102.692,A 0.000,B 0.000,C 90.000,E1 124.485} C_DIS
LIN {X 0.017,Y -315.440,Z 1102.691,A 0.000,B 0.000,C 90.000,E1 124.326} C_DIS
LIN {X 0.157,Y -318.532,Z 1102.689,A 0.000,B 0.000,C 90.000,E1 123.992} C_DIS
LIN {X 0.055,Y -322.129,Z 1102.686,A 0.000,B 0.000,C 90.000,E1 123.452} C_DIS
LIN {X -0.137,Y -323.563,Z 1102.684,A 0.000,B 0.000,C 90.000,E1 123.166} C_DIS
LIN {X -0.093,Y -335.326,Z 1102.667,A 0.000,B 0.000,C 90.000,E1 120.001} C_DIS
LIN {X -0.032,Y -347.302,Z 1102.651,A 0.000,B 0.000,C 90.000,E1 117.206} C_DIS
LIN {X 0.069,Y -360.740,Z 1102.636,A 0.000,B 0.000,C 90.000,E1 114.463} C_DIS
LIN {X 0.151,Y -374.013,Z 1102.623,A 0.000,B 0.000,C 90.000,E1 112.078} C_DIS
LIN {X 0.144,Y -388.631,Z 1102.610,A 0.000,B 0.000,C 90.000,E1 109.758} C_DIS
LIN {X 0.000,Y -404.696,Z 1102.597,A 0.000,B 0.000,C 90.000,E1 107.511} C_DIS
LIN {X -0.007,Y -422.325,Z 1102.585,A 0.000,B 0.000,C 90.000,E1 105.300} C_DIS
LIN {X -0.179,Y -441.589,Z 1102.573,A 0.000,B 0.000,C 90.000,E1 103.175} C_DIS
LIN {X 0.169,Y -461.747,Z 1102.562,A 0.000,B 0.000,C 90.000,E1 101.130} C_DIS
LIN {X 0.151,Y -466.873,Z 1102.559,A 0.000,B 0.000,C 90.000,E1 100.658} C_DIS
LIN {X 0.077,Y -469.242,Z 1102.558,A 0.000,B 0.000,C 90.000,E1 100.433} C_DIS
LIN {X -0.008,Y -471.108,Z 1102.557,A 0.000,B 0.000,C 90.000,E1 100.197} C_DIS
LIN {X -0.095,Y -472.520,Z 1102.555,A 0.000,B 0.000,C 90.000,E1 99.962} C_DIS
LIN {X 0.008,Y -474.385,Z 1102.552,A 0.000,B 0.000,C 90.000,E1 99.443} C_DIS
LIN {X 0.198,Y -475.147,Z 1102.550,A 0.000,B 0.000,C 90.000,E1 98.916} C_DIS
LIN {X -0.147,Y -474.938,Z 1102.547,A 0.000,B 0.000,C 90.000,E1 98.454} C_DIS
LIN {X -0.015,Y -473.730,Z 1102.544,A 0.000,B 0.000,C 90.000,E1 97.936} C_DIS
LIN {X -0.151,Y -472.696,Z 1102.543,A 0.000,B 0.000,C 90.000,E1 97.701} C_DIS
LIN {X 0.178,Y -471.307,Z 1102.541,A 0.000,B 0.000,C 90.000,E1 97.409} C_DIS
LIN {X 0.057,Y -456.857,Z 1102.530,A 0.000,B 0.000,C 90.000,E1 95.391} C_DIS
LIN {X 0.199,Y -440.925,Z 1102.517,A 0.000,B 0.000,C 90.000,E1 93.037} C_DIS
LIN {X 0.193,Y -427.893,Z 1102.505,A 0.000,B 0.000,C 90.000,E1 90.917} C_DIS
LIN {X -0.009,Y -413.970,Z 1102.492,A 0.000,B 0.000,C 90.000,E1 88.511} C_DIS
LIN {X 0.157,Y -403.603,Z 1102.481,A 0.000,B 0.000,C 90.000,E1 86.560} C_DIS
LIN {X 0.107,Y -392.996,Z 1102.470,A 0.000,B 0.000,C 90.000,E1 84.609} C_DIS
LIN {X -0.061,Y -380.837,Z 1102.458,A 0.000,B 0.000,C 90.000,E1 82.356} C_DIS
LIN {X -0.078,Y -371.571,Z 1102.448,A 0.000,B 0.000,C 90.000,E1 80.622} C_DIS
LIN {X -0.140,Y -361.953,Z 1102.438,A 0.000,B 0.000,C 90.000,E1 78.870} C_DIS
LIN {X -0.023,Y -352.086,Z 1102.428,A 0.000,B 0.000,C 90.000,E1 77.061} C_DIS
LIN {X -0.027,Y -340.486,Z 1102.416,A 0.000,B 0.000,C 90.000,E1 74.936} C_DIS
LIN {X 0.194,Y -327.494,Z 1102.402,A 0.000,B 0.000,C 90.000,E1 72.417} C_DIS
LIN {X -0.019,Y -310.652,Z 1102.383,A 0.000,B 0.000,C 90.000,E1 68.954} C_DIS
LIN {X -0.089,Y -299.184,Z 1102.369,A 0.000,B 0.000,C 90.000,E1 66.357} C_DIS
LIN {X -0.077,Y -288.033,Z 1102.354,A 0.000,B 0.000,C 90.000,E1 63.691} C_DIS
LIN {X -0.079,Y -277.196,Z 1102.339,A 0.000,B 0.000,C 90.000,E1 60.973} C_DIS
LIN {X -0.087,Y -266.634,Z 1102.323,A 0.000,B 0.000,C 90.000,E1 58.201} C_DIS
LIN {X 0.082,Y -255.198,Z 1102.306,A 0.000,B 0.000,C 90.000,E1 54.975} C_DIS
LIN {X -0.036,Y -244.389,Z 1102.287,A 0.000,B 0.000,C 90.000,E1 51.743} C_DIS
LIN {X 0.032,Y -235.454,Z 1102.271,A 0.000,B 0.000,C 90.000,E1 48.771} C_DIS
LIN {X -0.135,Y -227.135,Z 1102.254,A 0.000,B 0.000,C 90.000,E1 45.810} C_DIS
LIN {X 0.123,Y -219.172,Z 1102.237,A 0.000,B 0.000,C 90.000,E1 42.690} C_DIS
LIN {X 0.010,Y -209.831,Z 1102.216,A 0.000,B 0.000,C 90.000,E1 38.830} C_DIS
LIN {X -0.045,Y -202.783,Z 1102.198,A 0.000,B 0.000,C 90.000,E1 35.678} C_DIS
LIN {X -0.062,Y -196.328,Z 1102.180,A 0.000,B 0.000,C 90.000,E1 32.467} C_DIS
LIN {X -0.059,Y -190.494,Z 1102.162,A 0.000,B 0.000,C 90.000,E1 29.205} C_DIS
LIN {X -0.052,Y -185.287,Z 1102.144,A 0.000,B 0.000,C 90.000,E1 25.899} C_DIS
LIN {X 0.083,Y -180.837,Z 1102.125,A 0.000,B 0.000,C 90.000,E1 22.514} C_DIS
LIN {X 0.071,Y -177.063,Z 1102.106,A 0.000,B 0.000,C 90.000,E1 19.141} C_DIS
LIN {X 0.017,Y -173.275,Z 1102.083,A 0.000,B 0.000,C 90.000,E1 14.898} C_DIS
LIN {X 0.058,Y -170.156,Z 1102.054,A 0.000,B 0.000,C 90.000,E1 9.726} C_DIS
LIN {X 0.002,Y -168.096,Z 1102.011,A 0.000,B 0.000,C 90.000,E1 1.949} C_DIS
LIN {X -0.004,Y -169.786,Z 1101.959,A 0.000,B 0.000,C 90.000,E1 352.591} C_DIS
LIN {X -0.007,Y -172.643,Z 1101.930,A 0.000,B 0.000,C 90.000,E1 347.409} C_DIS
LIN {X -0.075,Y -176.150,Z 1101.906,A 0.000,B 0.000,C 90.000,E1 343.142} C_DIS
LIN {X 0.052,Y -180.640,Z 1101.883,A 0.000,B 0.000,C 90.000,E1 338.847} C_DIS
LIN {X 0.030,Y -185.007,Z 1101.864,A 0.000,B 0.000,C 90.000,E1 335.485} C_DIS
LIN {X 0.017,Y -190.099,Z 1101.845,A 0.000,B 0.000,C 90.000,E1 332.153} C_DIS
LIN {X -0.025,Y -195.981,Z 1101.827,A 0.000,B 0.000,C 90.000,E1 328.869} C_DIS
LIN {X 0.050,Y -202.491,Z 1101.809,A 0.000,B 0.000,C 90.000,E1 325.595} C_DIS
LIN {X 0.023,Y -209.796,Z 1101.791,A 0.000,B 0.000,C 90.000,E1 322.396} C_DIS
LIN {X 0.038,Y -218.942,Z 1101.771,A 0.000,B 0.000,C 90.000,E1 318.852} C_DIS
LIN {X -0.137,Y -228.004,Z 1101.754,A 0.000,B 0.000,C 90.000,E1 315.810} C_DIS
LIN {X -0.091,Y -238.178,Z 1101.738,A 0.000,B 0.000,C 90.000,E1 312.771} C_DIS
LIN {X -0.086,Y -248.254,Z 1101.723,A 0.000,B 0.000,C 90.000,E1 310.172} C_DIS
LIN {X 0.067,Y -261.371,Z 1101.707,A 0.000,B 0.000,C 90.000,E1 307.237} C_DIS
LIN {X 0.097,Y -275.769,Z 1101.691,A 0.000,B 0.000,C 90.000,E1 304.405} C_DIS
LIN {X 0.030,Y -291.403,Z 1101.676,A 0.000,B 0.000,C 90.000,E1 301.671} C_DIS
LIN {X 0.051,Y -308.176,Z 1101.661,A 0.000,B 0.000,C 90.000,E1 298.999} C_DIS
LIN {X -0.001,Y -328.899,Z 1101.645,A 0.000,B 0.000,C 90.000,E1 296.104} C_DIS
LIN {X -0.124,Y -343.883,Z 1101.635,A 0.000,B 0.000,C 90.000,E1 294.259} C_DIS
LIN {X -0.152,Y -361.900,Z 1101.624,A 0.000,B 0.000,C 90.000,E1 292.280} C_DIS
LIN {X 0.106,Y -375.430,Z 1101.616,A 0.000,B 0.000,C 90.000,E1 290.918} C_DIS
LIN {X 0.125,Y -394.692,Z 1101.607,A 0.000,B 0.000,C 90.000,E1 289.214} C_DIS
LIN {X 0.023,Y -408.032,Z 1101.600,A 0.000,B 0.000,C 90.000,E1 288.055} C_DIS
LIN {X 0.032,Y -418.573,Z 1101.595,A 0.000,B 0.000,C 90.000,E1 287.094} C_DIS
LIN {X -0.169,Y -426.288,Z 1101.591,A 0.000,B 0.000,C 90.000,E1 286.386} C_DIS
LIN {X -0.037,Y -433.792,Z 1101.587,A 0.000,B 0.000,C 90.000,E1 285.607} C_DIS
LIN {X 0.048,Y -440.922,Z 1101.582,A 0.000,B 0.000,C 90.000,E1 284.828} C_DIS
LIN {X -0.171,Y -447.743,Z 1101.578,A 0.000,B 0.000,C 90.000,E1 284.064} C_DIS
LIN {X 0.103,Y -453.918,Z 1101.574,A 0.000,B 0.000,C 90.000,E1 283.244} C_DIS
LIN {X 0.002,Y -459.438,Z 1101.569,A 0.000,B 0.000,C 90.000,E1 282.479} C_DIS
LIN {X -0.059,Y -464.306,Z 1101.565,A 0.000,B 0.000,C 90.000,E1 281.715} C_DIS
LIN {X -0.076,Y -468.443,Z 1101.561,A 0.000,B 0.000,C 90.000,E1 280.950} C_DIS
LIN {X -0.150,Y -471.940,Z 1101.557,A 0.000,B 0.000,C 90.000,E1 280.197} C_DIS
LIN {X 0.031,Y -473.907,Z 1101.554,A 0.000,B 0.000,C 90.000,E1 279.670} C_DIS
LIN {X 0.140,Y -475.614,Z 1101.551,A 0.000,B 0.000,C 90.000,E1 279.151} C_DIS
LIN {X -0.135,Y -477.035,Z 1101.548,A 0.000,B 0.000,C 90.000,E1 278.681} C_DIS
LIN {X -0.002,Y -478.213,Z 1101.545,A 0.000,B 0.000,C 90.000,E1 278.163} C_DIS
LIN {X 0.140,Y -479.177,Z 1101.543,A 0.000,B 0.000,C 90.000,E1 277.644} C_DIS
LIN {X -0.183,Y -479.896,Z 1101.540,A 0.000,B 0.000,C 90.000,E1 277.182} C_DIS
LIN {X -0.025,Y -480.350,Z 1101.537,A 0.000,B 0.000,C 90.000,E1 276.663} C_DIS
LIN {X 0.138,Y -480.479,Z 1101.534,A 0.000,B 0.000,C 90.000,E1 276.144} C_DIS
LIN {X -0.175,Y -480.330,Z 1101.531,A 0.000,B 0.000,C 90.000,E1 275.682} C_DIS
LIN {X -0.010,Y -479.855,Z 1101.529,A 0.000,B 0.000,C 90.000,E1 275.163} C_DIS
LIN {X 0.152,Y -478.970,Z 1101.526,A 0.000,B 0.000,C 90.000,E1 274.645} C_DIS
LIN {X -0.202,Y -477.660,Z 1101.523,A 0.000,B 0.000,C 90.000,E1 274.188} C_DIS
LIN {X -0.050,Y -475.843,Z 1101.520,A 0.000,B 0.000,C 90.000,E1 273.669} C_DIS
LIN {X 0.065,Y -473.373,Z 1101.518,A 0.000,B 0.000,C 90.000,E1 273.154} C_DIS
LIN {X 0.186,Y -470.153,Z 1101.515,A 0.000,B 0.000,C 90.000,E1 272.636} C_DIS
LIN {X -0.198,Y -466.014,Z 1101.512,A 0.000,B 0.000,C 90.000,E1 272.178} C_DIS
LIN {X 0.067,Y -463.543,Z 1101.510,A 0.000,B 0.000,C 90.000,E1 271.892} C_DIS
LIN {X -0.118,Y -460.728,Z 1101.509,A 0.000,B 0.000,C 90.000,E1 271.661} C_DIS
LIN {X -0.151,Y -457.824,Z 1101.508,A 0.000,B 0.000,C 90.000,E1 271.432} C_DIS
LIN {X 0.060,Y -451.461,Z 1101.505,A 0.000,B 0.000,C 90.000,E1 270.974} C_DIS
LIN {X -0.132,Y -444.728,Z 1101.503,A 0.000,B 0.000,C 90.000,E1 270.630} C_DIS
LIN {X 0.132,Y -437.685,Z 1101.502,A 0.000,B 0.000,C 90.000,E1 270.286} C_DIS
LIN {X -0.025,Y -430.414,Z 1101.500,A 0.000,B 0.000,C 90.000,E1 270.057} C_DIS
LIN {X 0.210,Y -423.074,Z 1101.499,A 0.000,B 0.000,C 90.000,E1 269.828} C_DIS
LIN {X -0.110,Y -415.474,Z 1101.498,A 0.000,B 0.000,C 90.000,E1 269.714} C_DIS
LIN {X -0.197,Y -407.329,Z 1101.498,A 0.000,B 0.000,C 90.000,E1 269.599} C_DIS
LIN {X -0.080,Y -397.062,Z 1101.497,A 0.000,B 0.000,C 90.000,E1 269.484} C_DIS
LIN {X 0.095,Y -388.877,Z 1101.497,A 0.000,B 0.000,C 90.000,E1 269.427} C_DIS
LIN {X 0.010,Y -181.421,Z 1101.497,A 0.000,B 0.000,C 90.000,E1 269.427} C_DIS
LIN {X -0.051,Y -180.830,Z 1101.472,A 0.000,B 0.000,C 90.000,E1 264.894} C_DIS
LIN {X 0.030,Y -178.935,Z 1101.443,A 0.000,B 0.000,C 90.000,E1 259.803} C_DIS
LIN {X 0.067,Y -175.984,Z 1101.415,A 0.000,B 0.000,C 90.000,E1 254.700} C_DIS
LIN {X 0.012,Y -175.480,Z 1101.410,A 0.000,B 0.000,C 90.000,E1 253.866} C_DIS
LIN {X 0.068,Y -172.226,Z 1101.387,A 0.000,B 0.000,C 90.000,E1 249.571} C_DIS
LIN {X 0.046,Y -171.703,Z 1101.382,A 0.000,B 0.000,C 90.000,E1 248.720} C_DIS
LIN {X -0.028,Y -167.298,Z 1101.353,A 0.000,B 0.000,C 90.000,E1 243.563} C_DIS
LIN {X 0.054,Y -166.676,Z 1101.348,A 0.000,B 0.000,C 90.000,E1 242.666} C_DIS
LIN {X -0.031,Y -162.657,Z 1101.324,A 0.000,B 0.000,C 90.000,E1 238.329} C_DIS
LIN {X 0.031,Y -161.347,Z 1101.314,A 0.000,B 0.000,C 90.000,E1 236.548} C_DIS
LIN {X 0.073,Y -157.341,Z 1101.290,A 0.000,B 0.000,C 90.000,E1 232.110} C_DIS
LIN {X 0.006,Y -155.327,Z 1101.275,A 0.000,B 0.000,C 90.000,E1 229.461} C_DIS
LIN {X -0.064,Y -151.679,Z 1101.250,A 0.000,B 0.000,C 90.000,E1 225.000} C_DIS
LIN {X -0.016,Y -150.543,Z 1101.240,A 0.000,B 0.000,C 90.000,E1 223.176} C_DIS
LIN {X 0.017,Y -147.268,Z 1101.215,A 0.000,B 0.000,C 90.000,E1 218.624} C_DIS
LIN {X -0.010,Y -145.296,Z 1101.194,A 0.000,B 0.000,C 90.000,E1 214.978} C_DIS
LIN {X -0.017,Y -142.392,Z 1101.164,A 0.000,B 0.000,C 90.000,E1 209.461} C_DIS
LIN {X 0.029,Y -141.371,Z 1101.148,A 0.000,B 0.000,C 90.000,E1 206.668} C_DIS
LIN {X 0.007,Y -139.346,Z 1101.112,A 0.000,B 0.000,C 90.000,E1 200.174} C_DIS
LIN {X 0.012,Y -139.018,Z 1101.102,A 0.000,B 0.000,C 90.000,E1 198.308} C_DIS
LIN {X 0.007,Y -138.342,Z 1101.055,A 0.000,B 0.000,C 90.000,E1 189.905} C_DIS
LIN {X 0.027,Y -139.393,Z 1101.008,A 0.000,B 0.000,C 90.000,E1 181.489} C_DIS
LIN {X -0.059,Y -141.292,Z 1100.972,A 0.000,B 0.000,C 90.000,E1 175.008} C_DIS
LIN {X 0.039,Y -142.654,Z 1100.957,A 0.000,B 0.000,C 90.000,E1 172.186} C_DIS
LIN {X -0.011,Y -144.995,Z 1100.931,A 0.000,B 0.000,C 90.000,E1 167.589} C_DIS
LIN {X -0.022,Y -147.622,Z 1100.911,A 0.000,B 0.000,C 90.000,E1 163.921} C_DIS
LIN {X 0.057,Y -150.249,Z 1100.890,A 0.000,B 0.000,C 90.000,E1 160.242} C_DIS
LIN {X 0.071,Y -153.644,Z 1100.870,A 0.000,B 0.000,C 90.000,E1 156.613} C_DIS
LIN {X -0.012,Y -157.059,Z 1100.850,A 0.000,B 0.000,C 90.000,E1 153.050} C_DIS
LIN {X 0.068,Y -161.189,Z 1100.830,A 0.000,B 0.000,C 90.000,E1 149.459} C_DIS
LIN {X 0.016,Y -163.283,Z 1100.821,A 0.000,B 0.000,C 90.000,E1 147.709} C_DIS
LIN {X 0.026,Y -167.726,Z 1100.801,A 0.000,B 0.000,C 90.000,E1 144.196} C_DIS
LIN {X -0.061,Y -171.544,Z 1100.787,A 0.000,B 0.000,C 90.000,E1 141.618} C_DIS
LIN {X -0.019,Y -176.487,Z 1100.768,A 0.000,B 0.000,C 90.000,E1 138.162} C_DIS
LIN {X 0.107,Y -180.785,Z 1100.753,A 0.000,B 0.000,C 90.000,E1 135.567} C_DIS
LIN {X -0.032,Y -186.192,Z 1100.735,A 0.000,B 0.000,C 90.000,E1 132.243} C_DIS
LIN {X 0.032,Y -190.829,Z 1100.721,A 0.000,B 0.000,C 90.000,E1 129.725} C_DIS
LIN {X -0.050,Y -196.588,Z 1100.703,A 0.000,B 0.000,C 90.000,E1 126.457} C_DIS
LIN {X -0.079,Y -200.122,Z 1100.693,A 0.000,B 0.000,C 90.000,E1 124.692} C_DIS
LIN {X 0.018,Y -308.157,Z 1100.693,A 0.000,B 0.000,C 90.000,E1 124.659} C_DIS
LIN {X 0.037,Y -310.385,Z 1100.692,A 0.000,B 0.000,C 90.000,E1 124.612} C_DIS
LIN {X -0.085,Y -315.816,Z 1100.691,A 0.000,B 0.000,C 90.000,E1 124.326} C_DIS
LIN {X 0.054,Y -318.750,Z 1100.689,A 0.000,B 0.000,C 90.000,E1 123.992} C_DIS
LIN {X 0.029,Y -320.762,Z 1100.687,A 0.000,B 0.000,C 90.000,E1 123.706} C_DIS
LIN {X 0.003,Y -322.337,Z 1100.686,A 0.000,B 0.000,C 90.000,E1 123.420} C_DIS
LIN {X 0.087,Y -323.702,Z 1100.684,A 0.000,B 0.000,C 90.000,E1 123.086} C_DIS
LIN {X -0.023,Y -335.456,Z 1100.666,A 0.000,B 0.000,C 90.000,E1 119.951} C_DIS
LIN {X -0.100,Y -347.451,Z 1100.651,A 0.000,B 0.000,C 90.000,E1 117.180} C_DIS
LIN {X -0.161,Y -360.910,Z 1100.636,A 0.000,B 0.000,C 90.000,E1 114.463} C_DIS
LIN {X -0.083,Y -374.202,Z 1100.623,A 0.000,B 0.000,C 90.000,E1 112.078} C_DIS
LIN {X -0.094,Y -388.841,Z 1100.610,A 0.000,B 0.000,C 90.000,E1 109.758} C_DIS
LIN {X 0.143,Y -404.929,Z 1100.597,A 0.000,B 0.000,C 90.000,E1 107.457} C_DIS
LIN {X 0.153,Y -422.582,Z 1100.585,A 0.000,B 0.000,C 90.000,E1 105.245} C_DIS
LIN {X 0.005,Y -441.866,Z 1100.573,A 0.000,B 0.000,C 90.000,E1 103.119} C_DIS
LIN {X -0.070,Y -462.033,Z 1100.562,A 0.000,B 0.000,C 90.000,E1 101.130} C_DIS
LIN {X -0.084,Y -467.161,Z 1100.559,A 0.000,B 0.000,C 90.000,E1 100.658} C_DIS
LIN {X -0.072,Y -469.457,Z 1100.558,A 0.000,B 0.000,C 90.000,E1 100.423} C_DIS
LIN {X 0.185,Y -471.290,Z 1100.557,A 0.000,B 0.000,C 90.000,E1 100.141} C_DIS
LIN {X 0.062,Y -472.670,Z 1100.555,A 0.000,B 0.000,C 90.000,E1 99.905} C_DIS
LIN {X 0.246,Y -474.443,Z 1100.552,A 0.000,B 0.000,C 90.000,E1 99.378} C_DIS
LIN {X -0.110,Y -475.131,Z 1100.549,A 0.000,B 0.000,C 90.000,E1 98.916} C_DIS
LIN {X 0.015,Y -474.850,Z 1100.547,A 0.000,B 0.000,C 90.000,E1 98.398} C_DIS
LIN {X 0.212,Y -473.563,Z 1100.544,A 0.000,B 0.000,C 90.000,E1 97.871} C_DIS
LIN {X 0.011,Y -472.482,Z 1100.542,A 0.000,B 0.000,C 90.000,E1 97.644} C_DIS
LIN {X -0.128,Y -471.033,Z 1100.541,A 0.000,B 0.000,C 90.000,E1 97.409} C_DIS
LIN {X 0.209,Y -456.558,Z 1100.530,A 0.000,B 0.000,C 90.000,E1 95.334} C_DIS
LIN {X -0.101,Y -440.652,Z 1100.517,A 0.000,B 0.000,C 90.000,E1 93.037} C_DIS
LIN {X -0.103,Y -427.628,Z 1100.505,A 0.000,B 0.000,C 90.000,E1 90.917} C_DIS
LIN {X 0.111,Y -413.726,Z 1100.491,A 0.000,B 0.000,C 90.000,E1 88.453} C_DIS
LIN {X -0.134,Y -403.368,Z 1100.481,A 0.000,B 0.000,C 90.000,E1 86.560} C_DIS
LIN {X -0.181,Y -392.757,Z 1100.470,A 0.000,B 0.000,C 90.000,E1 84.609} C_DIS
LIN {X 0.031,Y -380.586,Z 1100.457,A 0.000,B 0.000,C 90.000,E1 82.299} C_DIS
LIN {X 0.059,Y -372.868,Z 1100.449,A 0.000,B 0.000,C 90.000,E1 80.849} C_DIS
LIN {X -0.045,Y -363.246,Z 1100.439,A 0.000,B 0.000,C 90.000,E1 79.106} C_DIS
LIN {X 0.093,Y -353.411,Z 1100.430,A 0.000,B 0.000,C 90.000,E1 77.297} C_DIS
LIN {X 0.117,Y -341.808,Z 1100.418,A 0.000,B 0.000,C 90.000,E1 75.172} C_DIS
LIN {X -0.046,Y -328.772,Z 1100.404,A 0.000,B 0.000,C 90.000,E1 72.725} C_DIS
LIN {X 0.077,Y -311.838,Z 1100.385,A 0.000,B 0.000,C 90.000,E1 69.209} C_DIS
LIN {X -0.082,Y -298.910,Z 1100.368,A 0.000,B 0.000,C 90.000,E1 66.305} C_DIS
LIN {X -0.082,Y -287.750,Z 1100.354,A 0.000,B 0.000,C 90.000,E1 63.640} C_DIS
LIN {X -0.097,Y -276.907,Z 1100.338,A 0.000,B 0.000,C 90.000,E1 60.923} C_DIS
LIN {X 0.023,Y -266.338,Z 1100.323,A 0.000,B 0.000,C 90.000,E1 58.122} C_DIS
LIN {X -0.172,Y -254.882,Z 1100.305,A 0.000,B 0.000,C 90.000,E1 54.975} C_DIS
LIN {X -0.097,Y -244.063,Z 1100.287,A 0.000,B 0.000,C 90.000,E1 51.698} C_DIS
LIN {X 0.112,Y -235.126,Z 1100.271,A 0.000,B 0.000,C 90.000,E1 48.690} C_DIS
LIN {X -0.065,Y -226.792,Z 1100.254,A 0.000,B 0.000,C 90.000,E1 45.729} C_DIS
LIN {X -0.127,Y -218.815,Z 1100.237,A 0.000,B 0.000,C 90.000,E1 42.690} C_DIS
LIN {X 0.054,Y -209.441,Z 1100.215,A 0.000,B 0.000,C 90.000,E1 38.749} C_DIS
LIN {X -0.013,Y -202.364,Z 1100.198,A 0.000,B 0.000,C 90.000,E1 35.598} C_DIS
LIN {X 0.121,Y -195.928,Z 1100.180,A 0.000,B 0.000,C 90.000,E1 32.339} C_DIS
LIN {X 0.110,Y -190.089,Z 1100.162,A 0.000,B 0.000,C 90.000,E1 29.077} C_DIS
LIN {X 0.023,Y -184.924,Z 1100.143,A 0.000,B 0.000,C 90.000,E1 25.796} C_DIS
LIN {X -0.011,Y -180.484,Z 1100.125,A 0.000,B 0.000,C 90.000,E1 22.461} C_DIS
LIN {X -0.018,Y -175.886,Z 1100.101,A 0.000,B 0.000,C 90.000,E1 18.236} C_DIS
LIN {X 0.016,Y -172.359,Z 1100.078,A 0.000,B 0.000,C 90.000,E1 13.953} C_DIS
LIN {X -0.040,Y -169.486,Z 1100.049,A 0.000,B 0.000,C 90.000,E1 8.803} C_DIS
LIN {X 0.014,Y -170.304,Z 1099.949,A 0.000,B 0.000,C 90.000,E1 350.849} C_DIS
LIN {X 0.015,Y -173.005,Z 1099.925,A 0.000,B 0.000,C 90.000,E1 346.533} C_DIS
LIN {X 0.052,Y -176.695,Z 1099.901,A 0.000,B 0.000,C 90.000,E1 342.236} C_DIS
LIN {X 0.012,Y -180.378,Z 1099.882,A 0.000,B 0.000,C 90.000,E1 338.847} C_DIS
LIN {X -0.018,Y -184.750,Z 1099.864,A 0.000,B 0.000,C 90.000,E1 335.485} C_DIS
LIN {X -0.038,Y -189.873,Z 1099.845,A 0.000,B 0.000,C 90.000,E1 332.153} C_DIS
LIN {X -0.088,Y -195.760,Z 1099.827,A 0.000,B 0.000,C 90.000,E1 328.869} C_DIS
LIN {X -0.020,Y -202.286,Z 1099.809,A 0.000,B 0.000,C 90.000,E1 325.595} C_DIS
LIN {X -0.055,Y -209.599,Z 1099.791,A 0.000,B 0.000,C 90.000,E1 322.396} C_DIS
LIN {X -0.048,Y -218.800,Z 1099.771,A 0.000,B 0.000,C 90.000,E1 318.852} C_DIS
LIN {X 0.090,Y -227.835,Z 1099.754,A 0.000,B 0.000,C 90.000,E1 315.729} C_DIS
LIN {X 0.017,Y -236.683,Z 1099.739,A 0.000,B 0.000,C 90.000,E1 313.095} C_DIS
LIN {X 0.000,Y -246.606,Z 1099.725,A 0.000,B 0.000,C 90.000,E1 310.496} C_DIS
LIN {X -0.086,Y -259.542,Z 1099.709,A 0.000,B 0.000,C 90.000,E1 307.604} C_DIS
LIN {X -0.031,Y -275.712,Z 1099.691,A 0.000,B 0.000,C 90.000,E1 304.405} C_DIS
LIN {X -0.076,Y -289.388,Z 1099.678,A 0.000,B 0.000,C 90.000,E1 302.005} C_DIS
LIN {X -0.113,Y -305.993,Z 1099.663,A 0.000,B 0.000,C 90.000,E1 299.333} C_DIS
LIN {X -0.099,Y -326.572,Z 1099.647,A 0.000,B 0.000,C 90.000,E1 296.411} C_DIS
LIN {X -0.045,Y -341.457,Z 1099.636,A 0.000,B 0.000,C 90.000,E1 294.515} C_DIS
LIN {X -0.066,Y -359.887,Z 1099.625,A 0.000,B 0.000,C 90.000,E1 292.461} C_DIS
LIN {X 0.096,Y -375.909,Z 1099.616,A 0.000,B 0.000,C 90.000,E1 290.865} C_DIS
LIN {X -0.215,Y -395.164,Z 1099.607,A 0.000,B 0.000,C 90.000,E1 289.214} C_DIS
LIN {X -0.063,Y -408.730,Z 1099.600,A 0.000,B 0.000,C 90.000,E1 288.000} C_DIS
LIN {X -0.065,Y -419.287,Z 1099.595,A 0.000,B 0.000,C 90.000,E1 287.040} C_DIS
LIN {X -0.159,Y -426.988,Z 1099.591,A 0.000,B 0.000,C 90.000,E1 286.315} C_DIS
LIN {X -0.154,Y -434.502,Z 1099.586,A 0.000,B 0.000,C 90.000,E1 285.552} C_DIS
LIN {X -0.184,Y -441.664,Z 1099.582,A 0.000,B 0.000,C 90.000,E1 284.773} C_DIS
LIN {X 0.036,Y -448.459,Z 1099.578,A 0.000,B 0.000,C 90.000,E1 283.953} C_DIS
LIN {X -0.015,Y -454.585,Z 1099.573,A 0.000,B 0.000,C 90.000,E1 283.175} C_DIS
LIN {X -0.116,Y -460.077,Z 1099.569,A 0.000,B 0.000,C 90.000,E1 282.411} C_DIS
LIN {X -0.272,Y -464.901,Z 1099.565,A 0.000,B 0.000,C 90.000,E1 281.658} C_DIS
LIN {X 0.177,Y -468.962,Z 1099.560,A 0.000,B 0.000,C 90.000,E1 280.838} C_DIS
LIN {X 0.195,Y -472.384,Z 1099.556,A 0.000,B 0.000,C 90.000,E1 280.074} C_DIS
LIN {X -0.170,Y -474.299,Z 1099.553,A 0.000,B 0.000,C 90.000,E1 279.613} C_DIS
LIN {X -0.058,Y -475.947,Z 1099.551,A 0.000,B 0.000,C 90.000,E1 279.095} C_DIS
LIN {X 0.141,Y -477.372,Z 1099.548,A 0.000,B 0.000,C 90.000,E1 278.568} C_DIS
LIN {X -0.197,Y -478.523,Z 1099.545,A 0.000,B 0.000,C 90.000,E1 278.106} C_DIS
LIN {X -0.051,Y -479.455,Z 1099.542,A 0.000,B 0.000,C 90.000,E1 277.587} C_DIS
LIN {X 0.104,Y -480.182,Z 1099.539,A 0.000,B 0.000,C 90.000,E1 277.068} C_DIS
LIN {X -0.213,Y -480.592,Z 1099.536,A 0.000,B 0.000,C 90.000,E1 276.606} C_DIS
LIN {X -0.047,Y -480.720,Z 1099.534,A 0.000,B 0.000,C 90.000,E1 276.087} C_DIS
LIN {X 0.120,Y -480.494,Z 1099.531,A 0.000,B 0.000,C 90.000,E1 275.568} C_DIS
LIN {X -0.191,Y -480.013,Z 1099.528,A 0.000,B 0.000,C 90.000,E1 275.106} C_DIS
LIN {X -0.029,Y -479.091,Z 1099.526,A 0.000,B 0.000,C 90.000,E1 274.588} C_DIS
LIN {X 0.095,Y -477.729,Z 1099.523,A 0.000,B 0.000,C 90.000,E1 274.073} C_DIS
LIN {X -0.227,Y -475.814,Z 1099.520,A 0.000,B 0.000,C 90.000,E1 273.612} C_DIS
LIN {X 0.067,Y -474.654,Z 1099.519,A 0.000,B 0.000,C 90.000,E1 273.326} C_DIS
LIN {X 0.198,Y -471.722,Z 1099.516,A 0.000,B 0.000,C 90.000,E1 272.808} C_DIS
LIN {X -0.180,Y -467.976,Z 1099.513,A 0.000,B 0.000,C 90.000,E1 272.350} C_DIS
LIN {X -0.106,Y -463.103,Z 1099.510,A 0.000,B 0.000,C 90.000,E1 271.835} C_DIS
LIN {X 0.170,Y -460.257,Z 1099.509,A 0.000,B 0.000,C 90.000,E1 271.547} C_DIS
LIN {X 0.125,Y -453.987,Z 1099.506,A 0.000,B 0.000,C 90.000,E1 271.088} C_DIS
LIN {X 0.192,Y -447.346,Z 1099.504,A 0.000,B 0.000,C 90.000,E1 270.688} C_DIS
LIN {X -0.098,Y -440.552,Z 1099.502,A 0.000,B 0.000,C 90.000,E1 270.401} C_DIS
LIN {X 0.002,Y -433.357,Z 1099.501,A 0.000,B 0.000,C 90.000,E1 270.115} C_DIS
LIN {X 0.041,Y -425.605,Z 1099.499,A 0.000,B 0.000,C 90.000,E1 269.885} C_DIS
LIN {X 0.026,Y -417.703,Z 1099.498,A 0.000,B 0.000,C 90.000,E1 269.714} C_DIS
LIN {X -0.098,Y -409.946,Z 1099.498,A 0.000,B 0.000,C 90.000,E1 269.599} C_DIS
LIN {X -0.067,Y -399.565,Z 1099.497,A 0.000,B 0.000,C 90.000,E1 269.484} C_DIS
LIN {X 0.009,Y -389.873,Z 1099.497,A 0.000,B 0.000,C 90.000,E1 269.427} C_DIS
LIN {X -0.025,Y -181.418,Z 1099.497,A 0.000,B 0.000,C 90.000,E1 269.427} C_DIS
LIN {X 0.067,Y -180.824,Z 1099.471,A 0.000,B 0.000,C 90.000,E1 264.837} C_DIS
LIN {X -0.033,Y -178.928,Z 1099.443,A 0.000,B 0.000,C 90.000,E1 259.803} C_DIS
LIN {X 0.005,Y -175.975,Z 1099.415,A 0.000,B 0.000,C 90.000,E1 254.700} C_DIS
LIN {X -0.050,Y -175.463,Z 1099.410,A 0.000,B 0.000,C 90.000,E1 253.866} C_DIS
LIN {X 0.008,Y -172.213,Z 1099.386,A 0.000,B 0.000,C 90.000,E1 249.571} C_DIS
LIN {X -0.015,Y -171.689,Z 1099.382,A 0.000,B 0.000,C 90.000,E1 248.720} C_DIS
LIN {X -0.024,Y -167.916,Z 1099.358,A 0.000,B 0.000,C 90.000,E1 244.409} C_DIS
LIN {X -0.006,Y -166.658,Z 1099.348,A 0.000,B 0.000,C 90.000,E1 242.666} C_DIS
LIN {X 0.048,Y -162.642,Z 1099.324,A 0.000,B 0.000,C 90.000,E1 238.280} C_DIS
LIN {X -0.027,Y -161.330,Z 1099.314,A 0.000,B 0.000,C 90.000,E1 236.548} C_DIS
LIN {X 0.016,Y -157.325,Z 1099.290,A 0.000,B 0.000,C 90.000,E1 232.110} C_DIS
LIN {X -0.051,Y -155.307,Z 1099.275,A 0.000,B 0.000,C 90.000,E1 229.461} C_DIS
LIN {X -0.012,Y -151.664,Z 1099.250,A 0.000,B 0.000,C 90.000,E1 224.960} C_DIS
LIN {X 0.032,Y -150.530,Z 1099.240,A 0.000,B 0.000,C 90.000,E1 223.137} C_DIS
LIN {X -0.038,Y -147.255,Z 1099.214,A 0.000,B 0.000,C 90.000,E1 218.624} C_DIS
LIN {X 0.019,Y -145.281,Z 1099.194,A 0.000,B 0.000,C 90.000,E1 214.945} C_DIS
LIN {X 0.052,Y -142.384,Z 1099.163,A 0.000,B 0.000,C 90.000,E1 209.411} C_DIS
LIN {X -0.025,Y -141.361,Z 1099.148,A 0.000,B 0.000,C 90.000,E1 206.668} C_DIS
LIN {X -0.047,Y -139.342,Z 1099.112,A 0.000,B 0.000,C 90.000,E1 200.174} C_DIS
LIN {X -0.041,Y -139.012,Z 1099.102,A 0.000,B 0.000,C 90.000,E1 198.308} C_DIS
LIN {X -0.046,Y -138.341,Z 1099.055,A 0.000,B 0.000,C 90.000,E1 189.905} C_DIS
LIN {X -0.026,Y -139.398,Z 1099.008,A 0.000,B 0.000,C 90.000,E1 181.489} C_DIS
LIN {X 0.027,Y -141.302,Z 1098.972,A 0.000,B 0.000,C 90.000,E1 174.951} C_DIS
LIN {X -0.016,Y -142.663,Z 1098.957,A 0.000,B 0.000,C 90.000,E1 172.186} C_DIS
LIN {X -0.065,Y -145.009,Z 1098.931,A 0.000,B 0.000,C 90.000,E1 167.589} C_DIS
LIN {X -0.077,Y -147.636,Z 1098.911,A 0.000,B 0.000,C 90.000,E1 163.921} C_DIS
LIN {X 0.001,Y -150.266,Z 1098.890,A 0.000,B 0.000,C 90.000,E1 160.242} C_DIS
LIN {X 0.015,Y -153.666,Z 1098.870,A 0.000,B 0.000,C 90.000,E1 156.613} C_DIS
LIN {X 0.071,Y -157.082,Z 1098.850,A 0.000,B 0.000,C 90.000,E1 152.999} C_DIS
LIN {X 0.010,Y -161.217,Z 1098.830,A 0.000,B 0.000,C 90.000,E1 149.459} C_DIS
LIN {X -0.043,Y -163.306,Z 1098.821,A 0.000,B 0.000,C 90.000,E1 147.709} C_DIS
LIN {X -0.033,Y -167.754,Z 1098.801,A 0.000,B 0.000,C 90.000,E1 144.196} C_DIS
LIN {X -0.015,Y -171.571,Z 1098.786,A 0.000,B 0.000,C 90.000,E1 141.582} C_DIS
LIN {X -0.081,Y -176.518,Z 1098.767,A 0.000,B 0.000,C 90.000,E1 138.162} C_DIS
LIN {X 0.043,Y -180.817,Z 1098.753,A 0.000,B 0.000,C 90.000,E1 135.567} C_DIS
LIN {X 0.029,Y -186.226,Z 1098.734,A 0.000,B 0.000,C 90.000,E1 132.204} C_DIS
LIN {X -0.033,Y -190.863,Z 1098.721,A 0.000,B 0.000,C 90.000,E1 129.725} C_DIS
LIN {X 0.000,Y -196.625,Z 1098.702,A 0.000,B 0.000,C 90.000,E1 126.423} C_DIS
LIN {X 0.034,Y -200.055,Z 1098.693,A 0.000,B 0.000,C 90.000,E1 124.692} C_DIS
LIN {X 0.001,Y -307.301,Z 1098.693,A 0.000,B 0.000,C 90.000,E1 124.692} C_DIS
LIN {X 0.022,Y -309.532,Z 1098.693,A 0.000,B 0.000,C 90.000,E1 124.659} C_DIS
LIN {X 0.045,Y -313.562,Z 1098.692,A 0.000,B 0.000,C 90.000,E1 124.485} C_DIS
LIN {X -0.015,Y -315.845,Z 1098.691,A 0.000,B 0.000,C 90.000,E1 124.326} C_DIS
LIN {X -0.051,Y -318.980,Z 1098.689,A 0.000,B 0.000,C 90.000,E1 123.992} C_DIS
LIN {X -0.116,Y -320.956,Z 1098.687,A 0.000,B 0.000,C 90.000,E1 123.706} C_DIS
LIN {X 0.088,Y -322.500,Z 1098.686,A 0.000,B 0.000,C 90.000,E1 123.372} C_DIS
LIN {X -0.012,Y -324.918,Z 1098.682,A 0.000,B 0.000,C 90.000,E1 122.752} C_DIS
LIN {X -0.043,Y -335.564,Z 1098.666,A 0.000,B 0.000,C 90.000,E1 119.922} C_DIS
LIN {X 0.018,Y -347.574,Z 1098.651,A 0.000,B 0.000,C 90.000,E1 117.129} C_DIS
LIN {X 0.122,Y -361.049,Z 1098.636,A 0.000,B 0.000,C 90.000,E1 114.387} C_DIS
LIN {X 0.065,Y -374.359,Z 1098.622,A 0.000,B 0.000,C 90.000,E1 112.025} C_DIS
LIN {X 0.070,Y -389.014,Z 1098.609,A 0.000,B 0.000,C 90.000,E1 109.704} C_DIS
LIN {X -0.063,Y -405.122,Z 1098.597,A 0.000,B 0.000,C 90.000,E1 107.457} C_DIS
LIN {X -0.057,Y -422.796,Z 1098.585,A 0.000,B 0.000,C 90.000,E1 105.245} C_DIS
LIN {X -0.205,Y -442.097,Z 1098.573,A 0.000,B 0.000,C 90.000,E1 103.119} C_DIS
LIN {X 0.182,Y -462.272,Z 1098.562,A 0.000,B 0.000,C 90.000,E1 101.074} C_DIS
LIN {X 0.174,Y -467.401,Z 1098.559,A 0.000,B 0.000,C 90.000,E1 100.602} C_DIS
LIN {X 0.190,Y -469.631,Z 1098.558,A 0.000,B 0.000,C 90.000,E1 100.366} C_DIS
LIN {X -0.044,Y -471.436,Z 1098.556,A 0.000,B 0.000,C 90.000,E1 100.141} C_DIS
LIN {X -0.196,Y -472.791,Z 1098.555,A 0.000,B 0.000,C 90.000,E1 99.905} C_DIS
LIN {X -0.013,Y -474.491,Z 1098.552,A 0.000,B 0.000,C 90.000,E1 99.378} C_DIS
LIN {X 0.101,Y -475.118,Z 1098.549,A 0.000,B 0.000,C 90.000,E1 98.859} C_DIS
LIN {X -0.242,Y -474.780,Z 1098.547,A 0.000,B 0.000,C 90.000,E1 98.398} C_DIS
LIN {X -0.045,Y -473.428,Z 1098.544,A 0.000,B 0.000,C 90.000,E1 97.871} C_DIS
LIN {X 0.222,Y -472.305,Z 1098.542,A 0.000,B 0.000,C 90.000,E1 97.587} C_DIS
LIN {X 0.084,Y -470.807,Z 1098.541,A 0.000,B 0.000,C 90.000,E1 97.352} C_DIS
LIN {X -0.045,Y -456.318,Z 1098.530,A 0.000,B 0.000,C 90.000,E1 95.334} C_DIS
LIN {X 0.088,Y -440.420,Z 1098.517,A 0.000,B 0.000,C 90.000,E1 92.980} C_DIS
LIN {X -0.211,Y -425.785,Z 1098.503,A 0.000,B 0.000,C 90.000,E1 90.630} C_DIS
LIN {X -0.194,Y -407.627,Z 1098.485,A 0.000,B 0.000,C 90.000,E1 87.364} C_DIS
LIN {X -0.154,Y -397.133,Z 1098.474,A 0.000,B 0.000,C 90.000,E1 85.412} C_DIS
LIN {X 0.128,Y -386.444,Z 1098.463,A 0.000,B 0.000,C 90.000,E1 83.394} C_DIS
LIN {X 0.159,Y -377.317,Z 1098.454,A 0.000,B 0.000,C 90.000,E1 81.667} C_DIS
LIN {X 0.125,Y -367.853,Z 1098.444,A 0.000,B 0.000,C 90.000,E1 79.926} C_DIS
LIN {X -0.009,Y -358.081,Z 1098.434,A 0.000,B 0.000,C 90.000,E1 78.173} C_DIS
LIN {X 0.034,Y -346.479,Z 1098.423,A 0.000,B 0.000,C 90.000,E1 76.061} C_DIS
LIN {X -0.015,Y -333.337,Z 1098.409,A 0.000,B 0.000,C 90.000,E1 73.614} C_DIS
LIN {X 0.061,Y -316.050,Z 1098.390,A 0.000,B 0.000,C 90.000,E1 70.134} C_DIS
LIN {X 0.009,Y -302.904,Z 1098.374,A 0.000,B 0.000,C 90.000,E1 67.230} C_DIS
LIN {X -0.016,Y -291.651,Z 1098.359,A 0.000,B 0.000,C 90.000,E1 64.588} C_DIS
LIN {X -0.063,Y -280.702,Z 1098.344,A 0.000,B 0.000,C 90.000,E1 61.897} C_DIS
LIN {X 0.015,Y -270.013,Z 1098.328,A 0.000,B 0.000,C 90.000,E1 59.125} C_DIS
LIN {X 0.096,Y -259.638,Z 1098.313,A 0.000,B 0.000,C 90.000,E1 56.294} C_DIS
LIN {X -0.001,Y -248.459,Z 1098.295,A 0.000,B 0.000,C 90.000,E1 53.084} C_DIS
LIN {X -0.011,Y -238.089,Z 1098.277,A 0.000,B 0.000,C 90.000,E1 49.784} C_DIS
LIN {X -0.013,Y -228.510,Z 1098.258,A 0.000,B 0.000,C 90.000,E1 46.419} C_DIS
LIN {X -0.037,Y -220.472,Z 1098.241,A 0.000,B 0.000,C 90.000,E1 43.380} C_DIS
LIN {X 0.073,Y -212.779,Z 1098.224,A 0.000,B 0.000,C 90.000,E1 40.253} C_DIS
LIN {X -0.112,Y -205.502,Z 1098.206,A 0.000,B 0.000,C 90.000,E1 37.156} C_DIS
LIN {X 0.052,Y -198.712,Z 1098.188,A 0.000,B 0.000,C 90.000,E1 33.913} C_DIS
LIN {X 0.046,Y -192.561,Z 1098.170,A 0.000,B 0.000,C 90.000,E1 30.669} C_DIS
LIN {X 0.029,Y -187.043,Z 1098.152,A 0.000,B 0.000,C 90.000,E1 27.385} C_DIS
LIN {X -0.046,Y -182.276,Z 1098.134,A 0.000,B 0.000,C 90.000,E1 24.079} C_DIS
LIN {X 0.048,Y -178.218,Z 1098.115,A 0.000,B 0.000,C 90.000,E1 20.684} C_DIS
LIN {X 0.024,Y -174.039,Z 1098.091,A 0.000,B 0.000,C 90.000,E1 16.441} C_DIS
LIN {X -0.043,Y -170.967,Z 1098.068,A 0.000,B 0.000,C 90.000,E1 12.175} C_DIS
LIN {X 0.065,Y -168.350,Z 1098.034,A 0.000,B 0.000,C 90.000,E1 6.087} C_DIS
LIN {X -0.029,Y -169.293,Z 1097.959,A 0.000,B 0.000,C 90.000,E1 352.591} C_DIS
LIN {X -0.051,Y -172.104,Z 1097.930,A 0.000,B 0.000,C 90.000,E1 347.409} C_DIS
LIN {X 0.031,Y -175.606,Z 1097.906,A 0.000,B 0.000,C 90.000,E1 343.087} C_DIS
LIN {X -0.027,Y -180.121,Z 1097.882,A 0.000,B 0.000,C 90.000,E1 338.847} C_DIS
LIN {X -0.064,Y -184.503,Z 1097.864,A 0.000,B 0.000,C 90.000,E1 335.485} C_DIS
LIN {X 0.075,Y -189.649,Z 1097.845,A 0.000,B 0.000,C 90.000,E1 332.103} C_DIS
LIN {X 0.018,Y -195.542,Z 1097.827,A 0.000,B 0.000,C 90.000,E1 328.820} C_DIS
LIN {X -0.090,Y -202.079,Z 1097.809,A 0.000,B 0.000,C 90.000,E1 325.595} C_DIS
LIN {X 0.034,Y -209.403,Z 1097.791,A 0.000,B 0.000,C 90.000,E1 322.351} C_DIS
LIN {X -0.127,Y -218.651,Z 1097.771,A 0.000,B 0.000,C 90.000,E1 318.852} C_DIS
LIN {X 0.004,Y -227.693,Z 1097.754,A 0.000,B 0.000,C 90.000,E1 315.729} C_DIS
LIN {X -0.077,Y -236.527,Z 1097.739,A 0.000,B 0.000,C 90.000,E1 313.095} C_DIS
LIN {X 0.060,Y -246.487,Z 1097.725,A 0.000,B 0.000,C 90.000,E1 310.458} C_DIS
LIN {X -0.069,Y -257.733,Z 1097.711,A 0.000,B 0.000,C 90.000,E1 307.935} C_DIS
LIN {X -0.070,Y -273.774,Z 1097.693,A 0.000,B 0.000,C 90.000,E1 304.739} C_DIS
LIN {X 0.072,Y -287.376,Z 1097.679,A 0.000,B 0.000,C 90.000,E1 302.291} C_DIS
LIN {X 0.021,Y -306.012,Z 1097.663,A 0.000,B 0.000,C 90.000,E1 299.283} C_DIS
LIN {X 0.053,Y -326.611,Z 1097.646,A 0.000,B 0.000,C 90.000,E1 296.360} C_DIS
LIN {X 0.119,Y -341.525,Z 1097.636,A 0.000,B 0.000,C 90.000,E1 294.463} C_DIS
LIN {X 0.110,Y -360.205,Z 1097.625,A 0.000,B 0.000,C 90.000,E1 292.386} C_DIS
LIN {X 0.119,Y -376.566,Z 1097.616,A 0.000,B 0.000,C 90.000,E1 290.791} C_DIS
LIN {X 0.202,Y -395.820,Z 1097.606,A 0.000,B 0.000,C 90.000,E1 289.087} C_DIS
LIN {X -0.113,Y -409.375,Z 1097.600,A 0.000,B 0.000,C 90.000,E1 287.946} C_DIS
LIN {X -0.105,Y -419.917,Z 1097.594,A 0.000,B 0.000,C 90.000,E1 286.985} C_DIS
LIN {X -0.207,Y -427.604,Z 1097.590,A 0.000,B 0.000,C 90.000,E1 286.260} C_DIS
LIN {X -0.092,Y -435.105,Z 1097.586,A 0.000,B 0.000,C 90.000,E1 285.481} C_DIS
LIN {X 0.141,Y -442.271,Z 1097.582,A 0.000,B 0.000,C 90.000,E1 284.662} C_DIS
LIN {X 0.047,Y -449.041,Z 1097.577,A 0.000,B 0.000,C 90.000,E1 283.883} C_DIS
LIN {X -0.107,Y -455.141,Z 1097.573,A 0.000,B 0.000,C 90.000,E1 283.119} C_DIS
LIN {X -0.204,Y -460.614,Z 1097.568,A 0.000,B 0.000,C 90.000,E1 282.355} C_DIS
LIN {X 0.196,Y -465.394,Z 1097.564,A 0.000,B 0.000,C 90.000,E1 281.535} C_DIS
LIN {X 0.099,Y -469.419,Z 1097.560,A 0.000,B 0.000,C 90.000,E1 280.782} C_DIS
LIN {X 0.122,Y -472.769,Z 1097.556,A 0.000,B 0.000,C 90.000,E1 280.018} C_DIS
LIN {X -0.240,Y -474.653,Z 1097.553,A 0.000,B 0.000,C 90.000,E1 279.557} C_DIS
LIN {X -0.050,Y -476.280,Z 1097.550,A 0.000,B 0.000,C 90.000,E1 279.029} C_DIS
LIN {X 0.076,Y -477.654,Z 1097.547,A 0.000,B 0.000,C 90.000,E1 278.511} C_DIS
LIN {X 0.215,Y -478.787,Z 1097.545,A 0.000,B 0.000,C 90.000,E1 277.992} C_DIS
LIN {X -0.111,Y -479.713,Z 1097.542,A 0.000,B 0.000,C 90.000,E1 277.530} C_DIS
LIN {X 0.105,Y -480.382,Z 1097.539,A 0.000,B 0.000,C 90.000,E1 277.004} C_DIS
LIN {X 0.264,Y -480.835,Z 1097.536,A 0.000,B 0.000,C 90.000,E1 276.486} C_DIS
LIN {X -0.102,Y -480.945,Z 1097.533,A 0.000,B 0.000,C 90.000,E1 276.030} C_DIS
LIN {X 0.067,Y -480.726,Z 1097.531,A 0.000,B 0.000,C 90.000,E1 275.511} C_DIS
LIN {X -0.242,Y -480.208,Z 1097.528,A 0.000,B 0.000,C 90.000,E1 275.049} C_DIS
LIN {X -0.078,Y -479.242,Z 1097.525,A 0.000,B 0.000,C 90.000,E1 274.531} C_DIS
LIN {X 0.082,Y -477.848,Z 1097.522,A 0.000,B 0.000,C 90.000,E1 274.012} C_DIS
LIN {X 0.201,Y -475.886,Z 1097.520,A 0.000,B 0.000,C 90.000,E1 273.498} C_DIS
LIN {X -0.131,Y -473.255,Z 1097.517,A 0.000,B 0.000,C 90.000,E1 273.037} C_DIS
LIN {X -0.033,Y -469.867,Z 1097.514,A 0.000,B 0.000,C 90.000,E1 272.522} C_DIS
LIN {X 0.051,Y -465.463,Z 1097.511,A 0.000,B 0.000,C 90.000,E1 272.007} C_DIS
LIN {X -0.136,Y -462.891,Z 1097.510,A 0.000,B 0.000,C 90.000,E1 271.776} C_DIS
LIN {X 0.146,Y -457.017,Z 1097.507,A 0.000,B 0.000,C 90.000,E1 271.260} C_DIS
LIN {X 0.014,Y -450.589,Z 1097.505,A 0.000,B 0.000,C 90.000,E1 270.859} C_DIS
LIN {X -0.087,Y -443.910,Z 1097.503,A 0.000,B 0.000,C 90.000,E1 270.516} C_DIS
LIN {X -0.183,Y -436.807,Z 1097.501,A 0.000,B 0.000,C 90.000,E1 270.229} C_DIS
